(* CoDeSys 2.3.9.41 project: phase 8e.pro *)
(* Libraries: TcpIp.lib 21.3.13 08:03:14, TcBase.lib 14.5.09 12:14:08, TcSystem.lib 27.2.12 15:08:36, TcBaseMath.lib 27.7.04 12:07:56, TcMath.lib 23.9.04 15:15:30, TcMC2.lib 22.11.13 16:10:22, STANDARD.LIB 5.6.98 12:03:02, TcNC.lib 10.10.08 17:55:34, TcUtilities.lib 10.1.13 20:12:12, SysLibTargetVisu.lib 16.6.08 16:24:26, SysLibVisu.lib 7.7.04 18:17:22 *)

(* Task configuration *)
TASK Standard (PRIORITY := 1, INTERVAL := T#5ms);
	MAIN
END_TASK
TASK Fast (PRIORITY := 0, INTERVAL := T#1ms);
	MainFast();
END_TASK

(* Global variable list: Globale_Variablen *)
VAR_GLOBAL CONSTANT
	MAX_CSV_ROWS 			: UDINT := 150;
	MAX_CSV_COLUMNS 		: UDINT := 8;
	MAX_CSV_FIELD_LENGTH	: UDINT := 8;

END_VAR

VAR_GLOBAL
	FILEDATA1: ARRAY[0..MAX_CSV_ROWS, 0..MAX_CSV_COLUMNS ] OF STRING;
	trigger1: BOOL;			(* motor running*)
	trigger2: BOOL;			(* in velocity*)
	trigger3:BOOL;			(* vehicle moving*)
	encoderX:	ARRAY[1..6] OF		LREAL;
	encoderY:	ARRAY[1..6] OF		LREAL;
	heading:		ARRAY[1..6] OF		LREAL;
	headingA: LREAL;
	reset:		BOOL;
	home: BOOL;
	combinedX: LREAL;
	combinedY: LREAL;
	combinedH: LREAL;
(*for ROS*)
	robotPosX:	LREAL;
	robotPosY:	LREAL;
	robotPosTheta:	LREAL;
	robotVelX:	LREAL;
	robotVelY:	LREAL;
	robotVelTheta:	LREAL;
(*
###################
	TwinCAT NC Achsen
###################
*)


	Axis1 : AXIS_REF;
	PowerAxis1: MC_Power;
	MoveAxis1: MC_MoveVelocity;
	MoveAxis12: MC_MoveVelocity;
	ResetAxis1: MC_Reset;		(* debug function block output data *)
	HaltAxis1: MC_Halt;

	Axis2 : AXIS_REF;
	PowerAxis2: MC_Power;
	MoveAxis2: MC_MoveVelocity;
	MoveAxis22: MC_MoveVelocity;
	ResetAxis2: MC_Reset;		(* debug function block output data *)
	HaltAxis2: MC_Halt;

	Axis3 : AXIS_REF;
	PowerAxis3: MC_Power;
	MoveAxis3: MC_MoveVelocity;
	MoveAxis32: MC_MoveVelocity;
	ResetAxis3: MC_Reset;		(* debug function block output data *)
	HaltAxis3: MC_Halt;

	Axis4 : AXIS_REF;
	PowerAxis4: MC_Power;
	MoveAxis4: MC_MoveVelocity;
	MoveAxis42: MC_MoveVelocity;
	ResetAxis4: MC_Reset;		(* debug function block output data *)
	HaltAxis4: MC_Halt;


	LOCrobotPosX: LREAL;
	LOCrobotPosY: LREAL;
	LOCrobotPosTheta: LREAL;
	LOCrobotVelX: LREAL;
	LOCrobotVelY: LREAL;
	LOCrobotVelTheta: LREAL;
END_VAR

(* Global variable list: TwinCAT_Configuration *)
(* Generated automatically by TwinCAT - (read only) *)
VAR_CONFIG
	MainFast.fblocalization.encoder1.PlcToNc AT %QB1156 : PLCTONC_AXIS_REF;	(*  ~ {LinkedWith:TINC^NC-Task 1 SAF^Axes^encoder1^Inputs^encoder1_FromPlc} *)
	MainFast.fblocalization.encoder1.NcToPlc AT %IB1152 : NCTOPLC_AXIS_REF;	(*  ~ {LinkedWith:TINC^NC-Task 1 SAF^Axes^encoder1^Outputs^encoder1_ToPlc} *)
	MainFast.fblocalization.encoder2.PlcToNc AT %QB1284 : PLCTONC_AXIS_REF;	(*  ~ {LinkedWith:TINC^NC-Task 1 SAF^Axes^encoder2^Inputs^encoder2_FromPlc} *)
	MainFast.fblocalization.encoder2.NcToPlc AT %IB1280 : NCTOPLC_AXIS_REF;	(*  ~ {LinkedWith:TINC^NC-Task 1 SAF^Axes^encoder2^Outputs^encoder2_ToPlc} *)
	MainFast.fblocalization.encoder3.PlcToNc AT %QB1412 : PLCTONC_AXIS_REF;	(*  ~ {LinkedWith:TINC^NC-Task 1 SAF^Axes^encoder3^Inputs^encoder3_FromPlc} *)
	MainFast.fblocalization.encoder3.NcToPlc AT %IB1408 : NCTOPLC_AXIS_REF;	(*  ~ {LinkedWith:TINC^NC-Task 1 SAF^Axes^encoder3^Outputs^encoder3_ToPlc} *)
	MainFast.fblocalization.encoder4.PlcToNc AT %QB1540 : PLCTONC_AXIS_REF;	(*  ~ {LinkedWith:TINC^NC-Task 1 SAF^Axes^encoder4^Inputs^encoder4_FromPlc} *)
	MainFast.fblocalization.encoder4.NcToPlc AT %IB1536 : NCTOPLC_AXIS_REF;	(*  ~ {LinkedWith:TINC^NC-Task 1 SAF^Axes^encoder4^Outputs^encoder4_ToPlc} *)
	.Axis1.PlcToNc AT %QB1668 : PLCTONC_AXIS_REF;	(*  ~ {LinkedWith:TINC^NC-Task 1 SAF^Axes^motor 1^Inputs^motor 1_FromPlc} *)
	.Axis1.NcToPlc AT %IB1664 : NCTOPLC_AXIS_REF;	(*  ~ {LinkedWith:TINC^NC-Task 1 SAF^Axes^motor 1^Outputs^motor 1_ToPlc} *)
	.Axis2.PlcToNc AT %QB1796 : PLCTONC_AXIS_REF;	(*  ~ {LinkedWith:TINC^NC-Task 1 SAF^Axes^motor 2^Inputs^motor 2_FromPlc} *)
	.Axis2.NcToPlc AT %IB1792 : NCTOPLC_AXIS_REF;	(*  ~ {LinkedWith:TINC^NC-Task 1 SAF^Axes^motor 2^Outputs^motor 2_ToPlc} *)
	.Axis3.PlcToNc AT %QB1924 : PLCTONC_AXIS_REF;	(*  ~ {LinkedWith:TINC^NC-Task 1 SAF^Axes^motor 3^Inputs^motor 3_FromPlc} *)
	.Axis3.NcToPlc AT %IB1920 : NCTOPLC_AXIS_REF;	(*  ~ {LinkedWith:TINC^NC-Task 1 SAF^Axes^motor 3^Outputs^motor 3_ToPlc} *)
	.Axis4.PlcToNc AT %QB2052 : PLCTONC_AXIS_REF;	(*  ~ {LinkedWith:TINC^NC-Task 1 SAF^Axes^motor 4^Inputs^motor 4_FromPlc} *)
	.Axis4.NcToPlc AT %IB2048 : NCTOPLC_AXIS_REF;	(*  ~ {LinkedWith:TINC^NC-Task 1 SAF^Axes^motor 4^Outputs^motor 4_ToPlc} *)
END_VAR

(* Data type *)
TYPE MoveState_NC :
(
	NC_INIT,
	NC_ENABLE,
	NC_MOVE,
	NC_MOVENEXT,
	NC_ERROR,
	NC_RESET
);
END_TYPE

(* POU MAIN, ST *)
PROGRAM MAIN
VAR
	fbPLC_Reset: PLC_Reset;
	fbPLC_Start: PLC_Start;
	state_NC: MoveState_NC;
	Manual: BOOL := FALSE;
	bEnable: BOOL; (* gibt die Achse frei *)
	bReset_Axis: BOOL; (* Reset der Achse *)
	bAxis_Ready: ARRAY[1..5] OF	BOOL; (* Checks whether the axis is ready *)
	trigger2bypass: ARRAY[1..4] OF	BOOL;
	bMoveCombination: ARRAY[1..10] OF		BOOL; (* the combined movement *)
	i: INT;
	MotionReq: BOOL;
	timeToMove: TIME;
	directionToMove: INT;
	timeToMoveReal: LREAL;
	speedToMove: LREAL := 603;
	timeUp: BOOL;
	timerOn: BOOL;
	fbTON1: TON;
	myROS_connect_receiveData: ROS_connect_receiveData;
	myROS_connect_sendData: ROS_connect_sendData;
	myROS_disconnect: ROS_disconnect;
	myROS_receiveData: ROS_receiveData;
	myROS_sendData: ROS_sendData;
	myROS_convertSendData: ROS_convertSendData;
	ROS_tcpSocketReceiveData: T_HSOCKET;
	ROS_connectionOpenReceiveData: BOOL := FALSE;
	ROS_tcpSocketSendData: T_HSOCKET;
	ROS_connectionOpenSendData: BOOL := FALSE;
	ROS_closeConnection: BOOL := TRUE;
	ROS_velAxis1: LREAL := 0;
	ROS_velAxis2: LREAL := 0;
	ROS_velAxis3: LREAL := 0;
	ROS_velAxis4: LREAL := 0;
	ROS_RobotPosX: LREAL := 0;
	ROS_RobotPosY: LREAL := 0;
	ROS_RobotPosTheta: LREAL := 0;
	ROS_RobotVelX: LREAL := 0;
	ROS_RobotVelY: LREAL := 0;
	ROS_RobotVelTheta: LREAL := 0;
	sendBufferREAL: LREAL := 0;
	sendBuffer: STRING;
	sendTakt: LREAL := 0;
	vel_last1: LREAL;
	vel_current1: LREAL;
	vel_last2: LREAL;
	vel_current2: LREAL;
	vel_last3: LREAL;
	vel_current3: LREAL;
	vel_last4: LREAL;
	vel_current4: LREAL;
	startTimer1: BOOL;
	timer1On: BOOL;
	firstStart: BOOL;
	Q: BOOL;
	startPLC: BOOL;
	oldSpeedX: LREAL;
	oldSpeedY: LREAL;
	oldSpeedH: LREAL;
	connectJs: jsConnect;
	disconnectJs: jsDisconnect;
	receiveJsData: jsReceiveData;
	tcpSockeJst: T_HSOCKET;
	connectionOpen_js: BOOL := FALSE;
	closeConnection_js: BOOL := TRUE;
	XAxis: LREAL;
	YAxis: LREAL;
	ZAxis: LREAL;
	botton: LREAL;
	t1: INT;
	Name: BOOL;
END_VAR
(*
##
## This code was built by Theng Chua and Christian Scheifele, University of Stuttgart, 2014.
## It contains complete segments from Chris Jarrett, Auckland University, 2014
## and is derived in part from the TCP/IP server example on www.beckhoff.com
##
*)
(*IF (trigger3 = TRUE) THEN t1:=1; ELSE t1:=0; END_IF*)

(*
###################
Manual
###################
*)
IF (Manual=TRUE) THEN
	IF (reset=TRUE) THEN
	fbPLC_Reset(port:=801,RESET:=TRUE);
	fbPLC_Start(port:=801,start:=TRUE);
	(*set all globle variable to zero*)
	trigger1:=FALSE;
	trigger2:=FALSE;
	trigger3:=FALSE;
	home:= TRUE;
	combinedX:=0;
	combinedY:=0;
	combinedH:=0;
	END_IF

	FOR i:=1 TO 10 BY 1 DO
		IF(bMoveCombination[i]) THEN
			directionToMove:=i;
			MotionReq:=TRUE;
		END_IF
	END_FOR

	IF(MotionReq=TRUE) THEN
		CASE directionToMove OF
		1:	ROS_velAxis1:= -speedToMove;
			ROS_velAxis2:= 0;
			ROS_velAxis3:= 0;
			ROS_velAxis4:= -speedToMove;
		2:	ROS_velAxis1:= -speedToMove;
			ROS_velAxis2:= -speedToMove;
			ROS_velAxis3:= -speedToMove;
			ROS_velAxis4:= -speedToMove;
		3:	ROS_velAxis1:= 0;
			ROS_velAxis2:= -speedToMove;
			ROS_velAxis3:= -speedToMove;
			ROS_velAxis4:= 0;
		4:	ROS_velAxis1:= -speedToMove;
			ROS_velAxis2:= speedToMove;
			ROS_velAxis3:= speedToMove;
			ROS_velAxis4:= -speedToMove;
		5:	ROS_velAxis1:= speedToMove;
			ROS_velAxis2:= -speedToMove;
			ROS_velAxis3:= -speedToMove;
			ROS_velAxis4:= speedToMove;
		6:	ROS_velAxis1:= 0;
			ROS_velAxis2:= speedToMove;
			ROS_velAxis3:= speedToMove;
			ROS_velAxis4:= 0;
		7:	ROS_velAxis1:= speedToMove;
			ROS_velAxis2:= speedToMove;
			ROS_velAxis3:= speedToMove;
			ROS_velAxis4:= speedToMove;
		8:	ROS_velAxis1:= speedToMove;
			ROS_velAxis2:= 0;
			ROS_velAxis3:= 0;
			ROS_velAxis4:= speedToMove;
		9:	ROS_velAxis1:= -speedToMove;
			ROS_velAxis2:= speedToMove;
			ROS_velAxis3:= -speedToMove;
			ROS_velAxis4:= speedToMove;
		10:	ROS_velAxis1:= speedToMove;
			ROS_velAxis2:= -speedToMove;
			ROS_velAxis3:= speedToMove;
			ROS_velAxis4:= -speedToMove;
		ELSE
			ROS_velAxis1:= 0;
			ROS_velAxis2:= 0;
			ROS_velAxis3:= 0;
			ROS_velAxis4:= 0;
		END_CASE
	timetomove:= REAL_TO_TIME (timeToMoveReal);
	timerOn:=TRUE;
	END_IF

	fbTON1(IN:=timerOn, PT:=timeToMove, Q=>timeUp, ET=>);

	IF (timeUp=TRUE)  THEN
	MotionReq:=FALSE;
	bMoveCombination[directionToMove]:=FALSE;
	ROS_velAxis1:= 0;
	ROS_velAxis2:= 0;
	ROS_velAxis3:= 0;
	ROS_velAxis4:= 0;
	directionToMove:=0;
	timerOn:=FALSE;
	END_IF
(*
###################
ODOMETRY
###################
*) (* trigger 1 and trigger 2*)
	IF (vel_current1<>0 OR vel_current2<>0 OR vel_current3<>0 OR vel_current4<>0) THEN trigger1:=TRUE;
	ELSE trigger1:=FALSE;
	END_IF
	IF (trigger1) THEN  trigger2bypass[1]:=FALSE; trigger2bypass[2]:=FALSE; trigger2bypass[3]:=FALSE; trigger2bypass[4]:=FALSE;
		IF (vel_current1=0) THEN trigger2bypass[1]:=TRUE; END_IF
		IF (vel_current2=0) THEN trigger2bypass[2]:=TRUE;END_IF
		IF (vel_current3=0) THEN trigger2bypass[3]:=TRUE;END_IF
		IF (vel_current4=0) THEN trigger2bypass[4]:=TRUE;END_IF
	END_IF
	trigger2 := (MoveAxis1.InVelocity OR trigger2bypass[1]) AND (MoveAxis2.InVelocity OR trigger2bypass[2]) AND (MoveAxis3.InVelocity OR trigger2bypass[3]) AND (MoveAxis4.InVelocity OR trigger2bypass[4])
			OR  (MoveAxis12.InVelocity OR trigger2bypass[1]) AND (MoveAxis22.InVelocity OR trigger2bypass[2]) AND (MoveAxis32.InVelocity OR trigger2bypass[3]) AND (MoveAxis42.InVelocity OR trigger2bypass[4]);

ELSE  (* after this run on auto*)

(*###################
ROS TCP/IP CONNECTION
###################

Close TCP port from last time-remove after DEBUG*)

		IF ROS_closeConnection THEN
		myROS_disconnect(bCloseAll:=ROS_closeConnection);
		ROS_closeConnection:=FALSE;
		END_IF

		(*Open a connection to ROS - Receive Data*)
		IF NOT ROS_connectionOpenReceiveData THEN
		myROS_connect_receiveData(RosConnected=>ROS_connectionOpenReceiveData, socketToUse=>ROS_tcpSocketReceiveData);
		END_IF
		IF ROS_connectionOpenReceiveData THEN
		myROS_receiveData(socketToUse:=ROS_tcpSocketReceiveData,velAxis1=>ROS_velAxis1, velAxis2=>ROS_velAxis2, velAxis3=>ROS_velAxis3, velAxis4=>ROS_velAxis4);
		END_IF

		(*Open a connection to ROS - Send Data*)
		IF NOT ROS_connectionOpenSendData THEN
		myROS_connect_sendData(RosConnected=>ROS_connectionOpenSendData, socketToUse=>ROS_tcpSocketSendData);
		END_IF

		(*ODOMETRY SORCE*)
		ROS_RobotPosX := LOCrobotPosY;
		ROS_RobotPosY := LOCrobotPosX;
		ROS_RobotPosTheta :=  LOCrobotPosTheta;
		ROS_RobotVelX :=  LOCrobotVelX;
		ROS_RobotVelY :=  LOCrobotVelY;
		ROS_RobotVelTheta :=  LOCrobotVelTheta;

		IF ROS_connectionOpenSendData THEN
		(* TAKTZEIT EINSTELLEN *)
		sendTakt := sendTakt + 0.1;
			IF sendTakt > 1THEN
			myROS_convertSendData(robotPosX:=ROS_RobotPosX, robotPosY:=ROS_RobotPosY, robotPosTheta:= ROS_RobotPosTheta, robotVelX:=ROS_RobotVelX, robotVelY:=ROS_RobotVelY, robotVelTheta:=ROS_RobotVelTheta, send_message=>sendBuffer );
			myROS_sendData(sendBuffer:=sendBuffer, socketToUse:=ROS_tcpSocketSendData);
			sendTakt := 0;
			END_IF
		END_IF


END_IF (* for manual running*)

(*
###################
TwinCAT NC Achsen
###################
*)
Axis1.ReadStatus;
Axis2.ReadStatus;
Axis3.ReadStatus;
Axis4.ReadStatus;

vel_current1 := -ROS_velAxis1;
vel_current2 := ROS_velAxis2;
vel_current3 := -ROS_velAxis3;
vel_current4 := ROS_velAxis4;

(* move axis using a state machine *)
CASE state_NC OF
		NC_INIT :	(* initialisation *)
			(* initialize all function blocks *)
			MoveAxis1.Execute := FALSE;
			ResetAxis1.Execute := FALSE;
			MoveAxis2.Execute := FALSE;
			ResetAxis2.Execute := FALSE;
			MoveAxis3.Execute := FALSE;
			ResetAxis3.Execute := FALSE;
			MoveAxis4.Execute := FALSE;
			ResetAxis4.Execute := FALSE;
			MoveAxis12.Execute := FALSE;
			MoveAxis22.Execute := FALSE;
			MoveAxis32.Execute := FALSE;
			MoveAxis42.Execute := FALSE;
			HaltAxis1.Execute := FALSE;
			HaltAxis2.Execute := FALSE;
			HaltAxis3.Execute := FALSE;
			HaltAxis4.Execute := FALSE;

			state_NC := NC_ENABLE;

		NC_ENABLE :
			PowerAxis1.Enable := TRUE;
			PowerAxis1.Enable_Positive := TRUE;
			PowerAxis1.Enable_Negative := TRUE;
			PowerAxis2.Enable := TRUE;
			PowerAxis2.Enable_Positive := TRUE;
			PowerAxis2.Enable_Negative := TRUE;
			PowerAxis3.Enable := TRUE;
			PowerAxis3.Enable_Positive := TRUE;
			PowerAxis3.Enable_Negative := TRUE;
			PowerAxis4.Enable := TRUE;
			PowerAxis4.Enable_Positive := TRUE;
			PowerAxis4.Enable_Negative := TRUE;

			IF PowerAxis1.Status AND PowerAxis2.Status AND PowerAxis3.Status AND PowerAxis4.Status THEN
				state_NC := NC_MOVE;
			ELSIF PowerAxis1.Error AND PowerAxis2.Error AND PowerAxis3.Error AND PowerAxis4.Error THEN
				state_NC := NC_ERROR;
			END_IF

		NC_MOVE :
			IF vel_current1>0 THEN
				HaltAxis1.Execute := FALSE;
				MoveAxis1.Direction := MC_Positive_Direction;
				MoveAxis1.Velocity := vel_current1;
				MoveAxis1.BufferMode := MC_Aborting;
				MoveAxis1.Execute := TRUE;
			ELSIF vel_current1<0 THEN
				HaltAxis1.Execute := FALSE;
				MoveAxis1.Direction := MC_Negative_Direction;
				MoveAxis1.Velocity := -vel_current1;
				MoveAxis1.BufferMode := MC_Aborting;
				MoveAxis1.Execute := TRUE;
			ELSE
				HaltAxis1.BufferMode := MC_Aborting;
				HaltAxis1.Execute := TRUE;
			END_IF;


			IF vel_current2>0 THEN
				HaltAxis2.Execute := FALSE;
				MoveAxis2.Direction := MC_Positive_Direction;
				MoveAxis2.Velocity := vel_current2;
				MoveAxis2.BufferMode := MC_Aborting;
				MoveAxis2.Execute := TRUE;
			ELSIF vel_current2<0 THEN
				HaltAxis2.Execute := FALSE;
				MoveAxis2.Direction := MC_Negative_Direction;
				MoveAxis2.Velocity := -vel_current2;
				MoveAxis2.BufferMode := MC_Aborting;
				MoveAxis2.Execute := TRUE;
			ELSE
				HaltAxis2.BufferMode := MC_Aborting;
				HaltAxis2.Execute := TRUE;
			END_IF;


			IF vel_current3>0 THEN
				HaltAxis3.Execute := FALSE;
				MoveAxis3.Direction := MC_Positive_Direction;
				MoveAxis3.Velocity := vel_current3;
				MoveAxis3.BufferMode := MC_Aborting;
				MoveAxis3.Execute := TRUE;
			ELSIF vel_current3<0 THEN
				HaltAxis3.Execute := FALSE;
				MoveAxis3.Direction := MC_Negative_Direction;
				MoveAxis3.Velocity := -vel_current3;
				MoveAxis3.BufferMode := MC_Aborting;
				MoveAxis3.Execute := TRUE;
			ELSE
				HaltAxis3.BufferMode := MC_Aborting;
				HaltAxis3.Execute := TRUE;
			END_IF;


			IF vel_current4>0 THEN
				HaltAxis4.Execute := FALSE;
				MoveAxis4.Direction := MC_Positive_Direction;
				MoveAxis4.Velocity := vel_current4;
				MoveAxis4.BufferMode := MC_Aborting;
				MoveAxis4.Execute := TRUE;
			ELSIF vel_current4<0 THEN
				HaltAxis4.Execute := FALSE;
				MoveAxis4.Direction := MC_Negative_Direction;
				MoveAxis4.Velocity := -vel_current4;
				MoveAxis4.BufferMode := MC_Aborting;
				MoveAxis4.Execute := TRUE;
			ELSE
				HaltAxis4.BufferMode := MC_Aborting;
				HaltAxis4.Execute := TRUE;
			END_IF;

			IF vel_last1<>vel_current1 OR vel_last2<>vel_current2 OR vel_last3<>vel_current3 OR vel_last4<>vel_current4 THEN
				MoveAxis1.Execute := FALSE;
				MoveAxis2.Execute := FALSE;
				MoveAxis3.Execute := FALSE;
				MoveAxis4.Execute := FALSE;
				vel_last1 := vel_current1;
				vel_last2 := vel_current2;
				vel_last3 := vel_current3;
				vel_last4 := vel_current4;
				state_NC := NC_MOVENEXT;
			END_IF;
			IF  MoveAxis1.CommandAborted OR MoveAxis1.Error OR MoveAxis2.CommandAborted OR MoveAxis2.Error OR MoveAxis3.CommandAborted OR MoveAxis3.Error OR MoveAxis4.CommandAborted OR MoveAxis4.Error THEN
				state_NC := NC_MOVE;
			END_IF

		NC_MOVENEXT :
			IF vel_current1>0 THEN
				HaltAxis1.Execute := FALSE;
				MoveAxis12.Direction := MC_Positive_Direction;
				MoveAxis12.Velocity := vel_current1;
				MoveAxis12.BufferMode := MC_Aborting;
				MoveAxis12.Execute := TRUE;
			ELSIF vel_current1<0 THEN
				HaltAxis1.Execute := FALSE;
				MoveAxis12.Direction := MC_Negative_Direction;
				MoveAxis12.Velocity := -vel_current1;
				MoveAxis12.BufferMode := MC_Aborting;
				MoveAxis12.Execute := TRUE;
			ELSE
				HaltAxis1.BufferMode := MC_Aborting;
				HaltAxis1.Execute := TRUE;
			END_IF;


			IF vel_current2>0 THEN
				HaltAxis2.Execute := FALSE;
				MoveAxis22.Direction := MC_Positive_Direction;
				MoveAxis22.Velocity := vel_current2;
				MoveAxis22.BufferMode := MC_Aborting;
				MoveAxis22.Execute := TRUE;
			ELSIF vel_current2<0 THEN
				HaltAxis2.Execute := FALSE;
				MoveAxis22.Direction := MC_Negative_Direction;
				MoveAxis22.Velocity := -vel_current2;
				MoveAxis22.BufferMode := MC_Aborting;
				MoveAxis22.Execute := TRUE;
			ELSE
				HaltAxis2.BufferMode := MC_Aborting;
				HaltAxis2.Execute := TRUE;
			END_IF;


			IF vel_current3>0 THEN
				HaltAxis3.Execute := FALSE;
				MoveAxis32.Direction := MC_Positive_Direction;
				MoveAxis32.Velocity := vel_current3;
				MoveAxis32.BufferMode := MC_Aborting;
				MoveAxis32.Execute := TRUE;
			ELSIF vel_current3<0 THEN
				HaltAxis3.Execute := FALSE;
				MoveAxis32.Direction := MC_Negative_Direction;
				MoveAxis32.Velocity := -vel_current3;
				MoveAxis32.BufferMode := MC_Aborting;
				MoveAxis32.Execute := TRUE;
			ELSE
				HaltAxis3.BufferMode := MC_Aborting;
				HaltAxis3.Execute := TRUE;
			END_IF;


			IF vel_current4>0 THEN
				HaltAxis4.Execute := FALSE;
				MoveAxis42.Direction := MC_Positive_Direction;
				MoveAxis42.Velocity := vel_current4;
				MoveAxis42.BufferMode := MC_Aborting;
				MoveAxis42.Execute := TRUE;
			ELSIF vel_current4<0 THEN
				HaltAxis4.Execute := FALSE;
				MoveAxis42.Direction := MC_Negative_Direction;
				MoveAxis42.Velocity := -vel_current4;
				MoveAxis42.BufferMode := MC_Aborting;
				MoveAxis42.Execute := TRUE;
			ELSE
				HaltAxis4.BufferMode := MC_Aborting;
				HaltAxis4.Execute := TRUE;
			END_IF;

			IF vel_last1<>vel_current1 OR vel_last2<>vel_current2 OR vel_last3<>vel_current3 OR vel_last4<>vel_current4 THEN
				MoveAxis12.Execute := FALSE;
				MoveAxis22.Execute := FALSE;
				MoveAxis32.Execute := FALSE;
				MoveAxis42.Execute := FALSE;
				vel_last1 := vel_current1;
				vel_last2 := vel_current2;
				vel_last3 := vel_current3;
				vel_last4 := vel_current4;
				state_NC := NC_MOVE;
			END_IF;
			IF  MoveAxis12.CommandAborted OR MoveAxis12.Error OR MoveAxis22.CommandAborted OR MoveAxis22.Error OR MoveAxis32.CommandAborted OR MoveAxis32.Error OR MoveAxis42.CommandAborted OR MoveAxis42.Error THEN
				state_NC := NC_MOVE;
			END_IF


		NC_ERROR :
			IF Axis1.Status.Error OR Axis2.Status.Error OR Axis3.Status.Error OR Axis4.Status.Error THEN
				state_NC := NC_RESET;	(* axis error requires reset *)
			ELSE
				state_NC := NC_INIT;		(* function block errors don't need a reset *)
			END_IF

		NC_RESET :
			ResetAxis1.Execute := TRUE;
			ResetAxis2.Execute := TRUE;
			ResetAxis3.Execute := TRUE;
			ResetAxis4.Execute := TRUE;
			IF ResetAxis1.Done AND ResetAxis2.Done AND ResetAxis3.Done AND ResetAxis4.Done THEN
				state_NC := NC_INIT;
			ELSIF ResetAxis1.Error OR ResetAxis2.Error OR ResetAxis3.Error OR ResetAxis4.Error THEN
				state_NC := NC_INIT; (* can't do anything here *)
			END_IF

END_CASE

ActPower;	(* call the power function block *)
ActMove;	(* call the move function block *)
ActReset;	(* call the reset function block *)
ActHaltAxis1;
ActHaltAxis2;
ActHaltAxis3;
ActHaltAxis4;
END_PROGRAM
ACTION ActHaltAxis1:
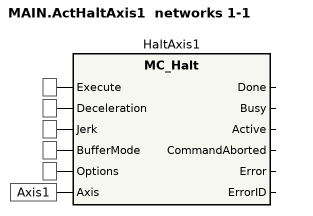
_FBD_ (* Function Block Diagram *)
NETWORK 1
	HaltAxis1:MC_Halt(Execute: , Deceleration: , Jerk: , BufferMode: , Options: , Axis: Axis1)
_END_FBD_
END_ACTION
ACTION ActHaltAxis2:
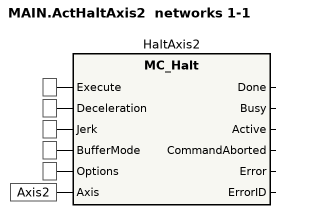
_FBD_ (* Function Block Diagram *)
NETWORK 1
	HaltAxis2:MC_Halt(Execute: , Deceleration: , Jerk: , BufferMode: , Options: , Axis: Axis2)
_END_FBD_
END_ACTION
ACTION ActHaltAxis3:
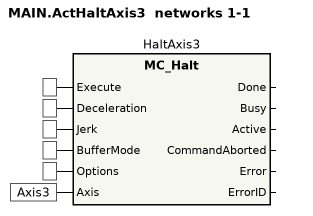
_FBD_ (* Function Block Diagram *)
NETWORK 1
	HaltAxis3:MC_Halt(Execute: , Deceleration: , Jerk: , BufferMode: , Options: , Axis: Axis3)
_END_FBD_
END_ACTION
ACTION ActHaltAxis4:
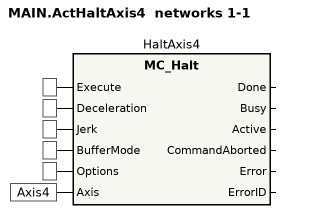
_FBD_ (* Function Block Diagram *)
NETWORK 1
	HaltAxis4:MC_Halt(Execute: , Deceleration: , Jerk: , BufferMode: , Options: , Axis: Axis4)
_END_FBD_
END_ACTION
ACTION ActMove:
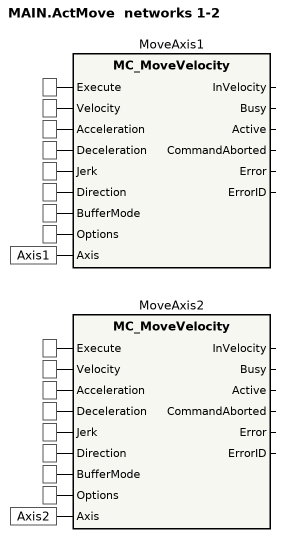
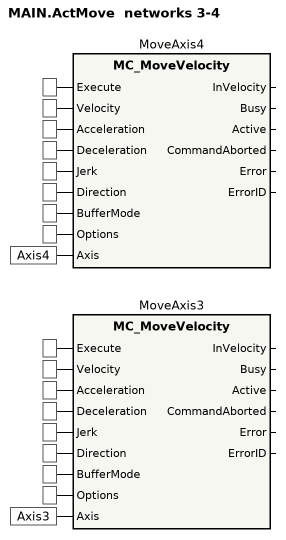
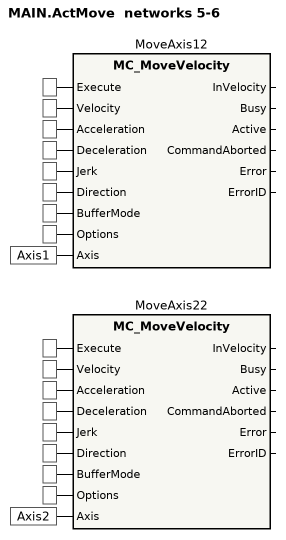
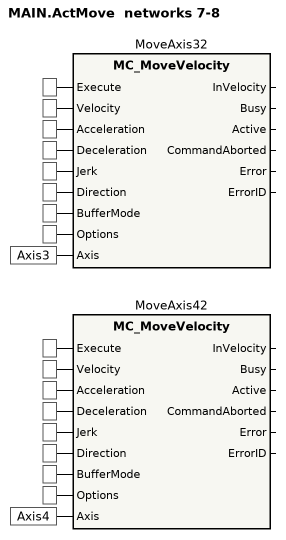
_FBD_ (* Function Block Diagram *)
NETWORK 1
	MoveAxis1:MC_MoveVelocity(Execute: , Velocity: , Acceleration: , Deceleration: , Jerk: , Direction: , BufferMode: , Options: , Axis: Axis1)
NETWORK 2
	MoveAxis2:MC_MoveVelocity(Execute: , Velocity: , Acceleration: , Deceleration: , Jerk: , Direction: , BufferMode: , Options: , Axis: Axis2)
NETWORK 3
	MoveAxis4:MC_MoveVelocity(Execute: , Velocity: , Acceleration: , Deceleration: , Jerk: , Direction: , BufferMode: , Options: , Axis: Axis4)
NETWORK 4
	MoveAxis3:MC_MoveVelocity(Execute: , Velocity: , Acceleration: , Deceleration: , Jerk: , Direction: , BufferMode: , Options: , Axis: Axis3)
NETWORK 5
	MoveAxis12:MC_MoveVelocity(Execute: , Velocity: , Acceleration: , Deceleration: , Jerk: , Direction: , BufferMode: , Options: , Axis: Axis1)
NETWORK 6
	MoveAxis22:MC_MoveVelocity(Execute: , Velocity: , Acceleration: , Deceleration: , Jerk: , Direction: , BufferMode: , Options: , Axis: Axis2)
NETWORK 7
	MoveAxis32:MC_MoveVelocity(Execute: , Velocity: , Acceleration: , Deceleration: , Jerk: , Direction: , BufferMode: , Options: , Axis: Axis3)
NETWORK 8
	MoveAxis42:MC_MoveVelocity(Execute: , Velocity: , Acceleration: , Deceleration: , Jerk: , Direction: , BufferMode: , Options: , Axis: Axis4)
_END_FBD_
END_ACTION
ACTION ActPower:
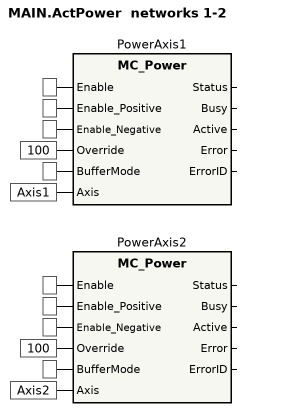
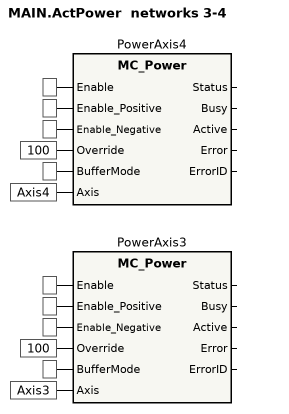
_FBD_ (* Function Block Diagram *)
NETWORK 1
	PowerAxis1:MC_Power(Enable: , Enable_Positive: , Enable_Negative: , Override: 100, BufferMode: , Axis: Axis1)
NETWORK 2
	PowerAxis2:MC_Power(Enable: , Enable_Positive: , Enable_Negative: , Override: 100, BufferMode: , Axis: Axis2)
NETWORK 3
	PowerAxis4:MC_Power(Enable: , Enable_Positive: , Enable_Negative: , Override: 100, BufferMode: , Axis: Axis4)
NETWORK 4
	PowerAxis3:MC_Power(Enable: , Enable_Positive: , Enable_Negative: , Override: 100, BufferMode: , Axis: Axis3)
_END_FBD_
END_ACTION
ACTION ActReset:
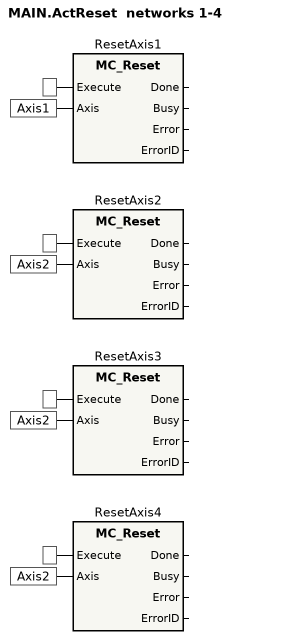
_FBD_ (* Function Block Diagram *)
NETWORK 1
	ResetAxis1:MC_Reset(Execute: , Axis: Axis1)
NETWORK 2
	ResetAxis2:MC_Reset(Execute: , Axis: Axis2)
NETWORK 3
	ResetAxis3:MC_Reset(Execute: , Axis: Axis2)
NETWORK 4
	ResetAxis4:MC_Reset(Execute: , Axis: Axis2)
_END_FBD_
END_ACTION

(* POU ROS_connect_receiveData, ST *)
FUNCTION_BLOCK ROS_connect_receiveData
VAR


	(*Functions*)
	openSocket: BOOL:=FALSE;
	fb_listen: FB_SocketListen;
	fb_accept: FB_SocketAccept;
	(*Timers*)
	fbAcceptTON: TON;

	(*TCP socket variables*)
	activeSocketHandle: T_HSOCKET;
	socketHandle: T_HSOCKET;



	(*Error variables*)
	listenError: UDINT:=0;
	acceptError: UDINT;
	listenErrSet: BOOL;
	closeError: UDINT;
	sendError: UDINT;
	receiveError: UDINT;
	bSendError: BOOL;


	(*Trigger Variables*)
	bCloseAll: BOOL := TRUE;

	(*Connection information*)
	portNumber: INT:=711;
	bAccepted: BOOL;

	(*Constants*)
	PLCPRJ_ACCEPT_POLLING_TIME: TIME:=T#1s;

	display: LREAL;
	heading: LREAL;

	state: INT:=0;

	xDist: LREAL;
	yDist: LREAL;
	zDist: LREAL;


	listening: BOOL;
END_VAR
VAR_OUTPUT
	RosConnected: BOOL;
	socketToUse: T_HSOCKET;
END_VAR
(*
##
## This code was built by Christian Scheifele, University of Stuttgart, 2014.
## It contains complete segments from Chris Jarrett, Auckland University, 2014
## and is derived in part from the TCP/IP server example on www.beckhoff.com
##
*)

CASE state OF
0:

IF(fb_Listen.hListener.localAddr.nPort=portNumber) THEN
RETURN;

ELSE
state:=1;
END_IF

1:
fb_listen
(
	sSrvNetId:='' ,
	sLocalHost:='',
	nLocalPort:=portNumber,
	bExecute:=TRUE,
	tTimeout:=T#5s,
	hListener=>socketHandle,
	nErrId=>listenError,
	bError=>listenErrSet,

);

	IF(fb_Listen.hListener.localAddr.nPort=portNumber) THEN
		fb_listen(bExecute:=FALSE); 		(*Start listening and move to the accept state*)

		state:=2;
	ELSE
		(*Return to the listening state*)
		state:=1;
	END_IF



2:

(*Start accepting a client connection*)
fbAcceptTON( IN := TRUE, PT := T#2s);  (*Start a timer to poll for the accepted connection*)
		IF fbAcceptTON.Q THEN
			fbAcceptTON( IN := FALSE );	(*Reset timer*)
			fb_accept(  bExecute := FALSE  ); (*Generate a rising edge to activate the accept function*)
			fb_accept(hListener := socketHandle, bExecute:= TRUE, hSocket=>activeSocketHandle );
			state:=3; (*Move to the state where the client is accepted*)

			fbAcceptTON( IN := FALSE);

		END_IF
3:
(*Complete accpeting the client connection*)
	fb_accept( bExecute := FALSE ); (*Reset the accept function to try connection again if necessary*)
	IF NOT fb_accept.bBusy THEN
		IF NOT fb_accept.bError THEN
			IF fb_accept.bAccepted THEN
				bAccepted := TRUE; (*If the client connection is accepted without error then move to the send state*)
				fb_accept(bExecute:=FALSE);
				socketToUse:=fb_accept.hSocket;
				state:=4;
			ELSE
				fb_listen(bExecute:=FALSE);
				fb_accept(bExecute:=FALSE);
				RosConnected:=FALSE; (*If the connection attempt was not successful, return the boolean as false*)
				fbAcceptTON( IN := FALSE);
				state:=2;
			END_IF
		END_IF
	END_IF
4:
RosConnected:=TRUE;
RETURN;

END_CASE;
END_FUNCTION_BLOCK

(* POU ROS_connect_sendData, ST *)
FUNCTION_BLOCK ROS_connect_sendData
VAR


	(*Functions*)
	openSocket: BOOL:=FALSE;
	fb_listen: FB_SocketListen;
	fb_accept: FB_SocketAccept;
	(*Timers*)
	fbAcceptTON: TON;

	(*TCP socket variables*)
	activeSocketHandle: T_HSOCKET;
	socketHandle: T_HSOCKET;



	(*Error variables*)
	listenError: UDINT:=0;
	acceptError: UDINT;
	listenErrSet: BOOL;
	closeError: UDINT;
	sendError: UDINT;
	receiveError: UDINT;
	bSendError: BOOL;


	(*Trigger Variables*)
	bCloseAll: BOOL := TRUE;

	(*Connection information*)
	portNumber: INT:=712;
	bAccepted: BOOL;

	(*Constants*)
	PLCPRJ_ACCEPT_POLLING_TIME: TIME:=T#1s;

	display: LREAL;
	heading: LREAL;

	state: INT:=0;

	xDist: LREAL;
	yDist: LREAL;
	zDist: LREAL;


	listening: BOOL;
END_VAR
VAR_OUTPUT
	RosConnected: BOOL;
	socketToUse: T_HSOCKET;
END_VAR
(*
##
## This code was built by Christian Scheifele, University of Stuttgart, 2014.
## It contains complete segments from Chris Jarrett, Auckland University, 2014
## and is derived in part from the TCP/IP server example on www.beckhoff.com
##
*)

CASE state OF
0:

IF(fb_Listen.hListener.localAddr.nPort=portNumber) THEN
RETURN;

ELSE
state:=1;
END_IF

1:
(*This code was built by Chris Jarrett, Auckland University, 2014. It is derived in part from the TCP/IP server example on www.beckhoff.com*)
fb_listen
(
	sSrvNetId:='' ,
	sLocalHost:='',
	nLocalPort:=portNumber,
	bExecute:=TRUE,
	tTimeout:=T#5s,
	hListener=>socketHandle,
	nErrId=>listenError,
	bError=>listenErrSet,

);

	IF(fb_Listen.hListener.localAddr.nPort=portNumber) THEN
		fb_listen(bExecute:=FALSE); 		(*Start listening and move to the accept state*)

		state:=2;
	ELSE
		(*Return to the listening state*)
		state:=1;
	END_IF



2:

(*Start accepting a client connection*)
fbAcceptTON( IN := TRUE, PT := T#2s);  (*Start a timer to poll for the accepted connection*)
		IF fbAcceptTON.Q THEN
			fbAcceptTON( IN := FALSE );	(*Reset timer*)
			fb_accept(  bExecute := FALSE  ); (*Generate a rising edge to activate the accept function*)
			fb_accept(hListener := socketHandle, bExecute:= TRUE, hSocket=>activeSocketHandle );
			state:=3; (*Move to the state where the client is accepted*)

			fbAcceptTON( IN := FALSE);

		END_IF
3:
(*Complete accpeting the client connection*)
	fb_accept( bExecute := FALSE ); (*Reset the accept function to try connection again if necessary*)
	IF NOT fb_accept.bBusy THEN
		IF NOT fb_accept.bError THEN
			IF fb_accept.bAccepted THEN
				bAccepted := TRUE; (*If the client connection is accepted without error then move to the send state*)
				fb_accept(bExecute:=FALSE);
				socketToUse:=fb_accept.hSocket;
				state:=4;
			ELSE
				fb_listen(bExecute:=FALSE);
				fb_accept(bExecute:=FALSE);
				RosConnected:=FALSE; (*If the connection attempt was not successful, return the boolean as false*)
				fbAcceptTON( IN := FALSE);
				state:=2;
			END_IF
		END_IF
	END_IF
4:
RosConnected:=TRUE;
RETURN;

END_CASE;
END_FUNCTION_BLOCK

(* POU ROS_disconnect, ST *)
FUNCTION_BLOCK ROS_disconnect
VAR_INPUT
	bCloseAll: BOOL;
END_VAR
VAR_OUTPUT
	connectionClosed: BOOL;
END_VAR
VAR
	fb_closeAll: FB_SocketCloseAll;
END_VAR
(*
##
## This code was built by Christian Scheifele, University of Stuttgart, 2014.
## It contains complete segments from Chris Jarrett, Auckland University, 2014
## and is derived in part from the TCP/IP server example on www.beckhoff.com
##
*)


(*This function closes the TCP/IP port being used the ROS connection*)

IF bCloseAll THEN
	bCloseAll:=FALSE;
	(*Close all open ports*)
	fb_closeAll(sSrvNetId:='', bExecute:=TRUE, tTimeOut:=T#5s );
ELSE
	fb_closeAll(bExecute:=FALSE);
END_IF


(*Move to the listening state*)
IF NOT fb_closeAll.bError THEN
	connectionClosed:=TRUE;


ELSE
connectionClosed:=FALSE;
END_IF
RETURN;
END_FUNCTION_BLOCK

(* POU ROS_receiveData, ST *)
FUNCTION_BLOCK ROS_receiveData
VAR_INPUT
	socketToUse: T_HSOCKET;
END_VAR
VAR_OUTPUT
	dataReceived: BOOL;
	velAxis1: LREAL;
	velAxis2: LREAL;
	velAxis3: LREAL;
	velAxis4: LREAL;
END_VAR
VAR
	(*Connection timers*)
	fbReceiveTON: TON;
	fbResetTON:TON;
	reset: BOOL;
	timeup:BOOL;

 	(*Functions*)
	fb_receive: FB_SocketReceive;

	(*Send and receive data and variables*)
	receiveBuffer: ARRAY[0..27] OF BYTE;
	bytesReceived: UDINT;
	sendBuffer: STRING;
	sendBufferAddress: DWORD;
	cbReceived, startPos, endPos, idx : UDINT;
	cbFrame: UDINT;
	sFromClient: T_MaxString;
	overflow: BOOL;
	endFound: BOOL;

	(*Error variables*)
	acceptError: UDINT;
	receiveError: UDINT;

	state: INT:=1;
END_VAR
(*
##
## This code was built by Christian Scheifele, University of Stuttgart, 2014.
## It contains complete segments from Chris Jarrett, Auckland University, 2014
## and is derived in part from the TCP/IP server example on www.beckhoff.com
##
*)

CASE state OF
1:
(*Receive information*)
	fbReceiveTON(  IN := FALSE, PT:=T#0s); (*Receive first request immediately*)
	fbReceiveTON(  IN := TRUE ); (*Start a timer to ensure complete transfer of information*)

		IF fbReceiveTON.Q THEN
			fbReceiveTON(  IN := FALSE);
			fb_receive(bExecute:=FALSE);  (*Generate a rising edge to start receiving data*)
			fb_receive
			(
				sSrvNetId:='',
				hSocket :=socketToUse,
				cbLen:=SIZEOF(receiveBuffer)-cbReceived,
				pDest:=ADR(receiveBuffer)+cbReceived,
				tTimeout:=T#5s,
				nRecBytes=>bytesReceived,
				nErrId=>receiveError,
				bExecute:=TRUE,
			);

	(*Move to the receive completion state*)
	state:=2;
	END_IF

2:
(*Continue receiving data*)
	fb_receive( bExecute := FALSE );
	IF NOT fb_receive.bBusy THEN
		IF NOT fb_receive.bError THEN (*If no error has occurred then start the actual receiving of data*)

			IF (fb_receive.nRecBytes>0) THEN (*Bytes have been received*)

				startPos:=cbReceived; (*index of first data byte*)
				endPos:=cbReceived+fb_receive.nRecBytes-1; (*index of last byte*)
				cbReceived:=cbReceived+fb_receive.nRecBytes; (*Calculating the number of received data bytes*)
				cbFrame:=0; (*Reset the frame length*)


				IF cbReceived<SIZEOF(sFromClient) THEN (*no overflow*)
					fbReceiveTON(IN:=FALSE, PT:=T#0S);

					(*Search for the string delimiter(separation character for different strings)*)
					FOR idx:=startPos TO endPos BY 1 DO
						IF receiveBuffer[idx]=0 THEN (*String delimiter found*)
							cbFrame:=idx+1;(*calculate length of received string*)
							MEMCPY(ADR(sFromClient), ADR(receiveBuffer),cbFrame); (*copy the received string to the output variable*)
							MEMMOVE(ADR(receiveBuffer), ADR(receiveBuffer[cbFrame]), cbReceived-cbFrame);(*move remaining data bytes*)
							dataReceived:=TRUE;  	(*Send an acknowledgement of data received*)
							state:=3; (*Move to the receive completion state*)
							endFound:=TRUE;
							EXIT;
						END_IF
					END_FOR
				ELSE(*no more free buffer space-overflow*)

					dataReceived:=FALSE;; (*Go to error state*)
					overflow:=TRUE;
					state:=4;
				END_IF
			ELSE(*no data received*)
					fbReceiveTON(IN:=FALSE, PT:=T#0ms);
					state:=1;
			END_IF
		ELSE(*error receiving data, exit function*)
			state:=4;
			dataReceived:=FALSE;
		END_IF
	END_IF

3:
(*State used to process data*)
	velAxis1:=(STRING_TO_LREAL(MID(sFromClient, 7, 1)))/100;  (*Extract the x distance*)
	velAxis2:=(STRING_TO_LREAL(MID(sFromClient, 7, 8)))/100;
	velAxis3:=(STRING_TO_LREAL(MID(sFromClient, 7, 15)))/100;
	velAxis4:=(STRING_TO_LREAL(MID(sFromClient, 7, 22)))/100;

       (*Fixing an issue of negative numbers
	IF velAxis1 >  -100 THEN
		velAxis1:=velAxis1/10;
	END_IF
	IF velAxis2 > -100 THEN
		velAxis2:=velAxis2/10;
	END_IF
	IF velAxis3 > -100 THEN
		velAxis3:=velAxis3/10;
	END_IF
	IF velAxis4 > -100  THEN
		velAxis4:=velAxis4/10;
	END_IF*)

	fb_receive(bExecute:=FALSE); (*Reset the receive function*)
	startPos:=0; (*reset buffer beginning pointer*)
	endPos:=0;  (*reset buffer end pointer*)
	cbReceived:=0; (*reset bytes received counter*)
	sFromClient:=''; (*reset transition variable*)

	state:=1;
	RETURN;

4: (*Unused except for as an error state*)
	trigger1:=FALSE;trigger2:=TRUE;
	trigger2:=FALSE;

	velAxis1:=0;
	velAxis2:=0;
	velAxis3:=0;
	velAxis4:=0;

	(*Clear buffer-PROBABLY UNNECESSARY*)
	receiveBuffer[0]:=0;
	receiveBuffer[1]:=0;
	receiveBuffer[2]:=0;
	receiveBuffer[3]:=0;
	receiveBuffer[4]:=0;
	receiveBuffer[5]:=0;
	receiveBuffer[6]:=0;
	receiveBuffer[7]:=0;
	receiveBuffer[8]:=0;
	receiveBuffer[9]:=0;
	receiveBuffer[10]:=0;
	receiveBuffer[11]:=0;
	receiveBuffer[12]:=0;
	receiveBuffer[13]:=0;
	receiveBuffer[14]:=0;
	receiveBuffer[15]:=0;
	receiveBuffer[16]:=0;
	receiveBuffer[17]:=0;
	receiveBuffer[18]:=0;
	receiveBuffer[19]:=0;
	receiveBuffer[20]:=0;
	receiveBuffer[21]:=0;
	receiveBuffer[22]:=0;
	receiveBuffer[23]:=0;
	receiveBuffer[24]:=0;
	receiveBuffer[25]:=0;
	receiveBuffer[26]:=0;
	receiveBuffer[27]:=0;

	state:=1;
END_CASE;
END_FUNCTION_BLOCK

(* POU ROS_sendData, ST *)
FUNCTION_BLOCK ROS_sendData
VAR_INPUT
	sendBuffer: STRING;
	socketToUse: T_HSOCKET;
END_VAR
VAR_OUTPUT
END_VAR
VAR
 	(*Functions*)
	fb_send1: FB_SocketSend;
	(*Send data and variables*)
	sendBufferAddress1: DWORD;
	sendError1: UDINT;
END_VAR
(*
##
## This code was built by Christian Scheifele, University of Stuttgart, 2014.
## It  is derived in part from the TCP/IP server example on www.beckhoff.com
##
*)
	(*Send a greeting to the client*)
	sendBufferAddress1:=ADR(sendBuffer);
	(*Send information*)
	fb_send1
	(
		sSrvNetId:='',
		hSocket:=socketToUse,
		cbLen:=INT_TO_UDINT(LEN( sendBuffer ))+1,
		pSrc:=sendBufferAddress1,
		bExecute:=TRUE,
		tTimeout:=T#5s,
		nErrId=>sendError1,
	);

	fb_send1( bExecute := FALSE );
	fb_send1( bExecute := TRUE );
	fb_send1( bExecute := FALSE );
END_FUNCTION_BLOCK

(* POU ROS_convertSendData, ST *)
FUNCTION_BLOCK ROS_convertSendData
VAR_INPUT
	robotPosX: LREAL;
	robotPosY: LREAL;
	robotPosTheta: LREAL;
	robotVelX: LREAL;
	robotVelY: LREAL;
	robotVelTheta: LREAL;
END_VAR
VAR_OUTPUT
	send_message: STRING;
END_VAR
VAR
	posXString: STRING;
	posYString: STRING;
	posThetaString: STRING;
	velXString: STRING;
	velYString: STRING;
	velThetaString: STRING;
END_VAR
(*
##
## This code was built by Christian Scheifele, University of Stuttgart, 2014.
##
*)

(* Eingangsdaten verarbeiten *)
posXString := LREAL_TO_STRING(ABS(robotPosX));
posYString := LREAL_TO_STRING(ABS(robotPosY));
posThetaString := LREAL_TO_STRING(ABS(robotPosTheta)*100);
velXString := LREAL_TO_STRING(ABS(robotVelX));
velYString := LREAL_TO_STRING(ABS(robotVelY));
velThetaString := LREAL_TO_STRING(ABS(robotVelTheta)*100);

(* posXString bearbeiten *)
posXString := LEFT(posXString, FIND(posXString, '.')-1);
IF LEN(posXString) < 6 THEN
posXString := INSERT(posXString, '0000000',0 );
posXString := RIGHT(posXString, 5);
IF(robotPosX < 0) THEN
posXString := INSERT(posXString, '-',0 );
ELSE
posXString := INSERT(posXString, '0',0 );
END_IF;
END_IF;


(* posYString bearbeiten *)
posYString := LEFT(posYString, FIND(posYString, '.')-1);
IF LEN(posYString) < 7 THEN
	posYString := INSERT(posYString, '0000000',0 );
	posYString := RIGHT(posYString, 6);
	IF(robotPosY < 0) THEN
		posYString := INSERT(posYString, '-',0 );
	ELSE
		posYString := INSERT(posYString, '0',0 );
	END_IF;
END_IF;

(* posThetaString bearbeiten *)
posThetaString := LEFT(posThetaString, FIND(posThetaString, '.')-1);
IF LEN(posThetaString) < 7 THEN
	posThetaString := INSERT(posThetaString, '0000000',0 );
	posThetaString := RIGHT(posThetaString, 6);
	IF(robotPosTheta < 0) THEN
		posThetaString := INSERT(posThetaString, '-',0 );
	ELSE
		posThetaString := INSERT(posThetaString, '0',0 );
	END_IF;
END_IF;

(* velXString bearbeiten *)
velXString := LEFT(velXString, FIND(velXString, '.')-1);
IF LEN(velXString) < 7 THEN
velXString := INSERT(velXString, '0000000',0 );
velXString := RIGHT(velXString, 6);
	IF(robotVelX < 0) THEN
		velXString := INSERT(velXString, '-',0 );
	ELSE
		velXString := INSERT(velXString, '0',0 );
	END_IF;
END_IF;

(* velYString bearbeiten *)
velYString := LEFT(velYString, FIND(velYString, '.')-1);
IF LEN(velYString) < 7 THEN
velYString := INSERT(velYString, '0000000',0 );
velYString := RIGHT(velYString, 6);
	IF(robotVelY < 0) THEN
		velYString := INSERT(velYString, '-',0 );
	ELSE
		velYString := INSERT(velYString, '0',0 );
	END_IF;
END_IF;

(* velThetaString bearbeiten *)
velThetaString := LEFT(velThetaString, FIND(velThetaString, '.')-1);
IF LEN(velThetaString) < 7 THEN
velThetaString := INSERT(velThetaString, '0000000',0 );
velThetaString := RIGHT(velThetaString, 6);
	IF(robotVelTheta < 0) THEN
		velThetaString := INSERT(velThetaString, '-',0 );
	ELSE
		velThetaString := INSERT(velThetaString, '0',0 );
	END_IF;
END_IF;

send_message := CONCAT (posXString, ' ');
send_message := CONCAT (send_message, posYString);
send_message := CONCAT (send_message, ' ');
send_message := CONCAT (send_message, posThetaString);
send_message := CONCAT (send_message, ' ');
send_message := CONCAT (send_message, velXString);
send_message := CONCAT (send_message, ' ');
send_message := CONCAT (send_message, velYString);
send_message := CONCAT (send_message, ' ');
send_message := CONCAT (send_message, velThetaString);

(*send_message := '-000001 0000002 0009000 0000009 -000001 0000004';*)
END_FUNCTION_BLOCK

(* POU jsConnect, ST *)
FUNCTION_BLOCK jsConnect
VAR


	(*Functions*)
	openSocket: BOOL:=FALSE;
	fb_listen: FB_SocketListen;
	fb_accept: FB_SocketAccept;
	(*Timers*)
	fbAcceptTON: TON;

	(*TCP socket variables*)
	activeSocketHandle: T_HSOCKET;
	socketHandle: T_HSOCKET;



	(*Error variables*)
	listenError: UDINT:=0;
	acceptError: UDINT;
	listenErrSet: BOOL;
	closeError: UDINT;
	sendError: UDINT;
	receiveError: UDINT;
	bSendError: BOOL;


	(*Trigger Variables*)
	bCloseAll: BOOL := TRUE;

	(*Connection information*)
	portNumber: INT:=8880;
	bAccepted: BOOL;

	(*Constants*)
	PLCPRJ_ACCEPT_POLLING_TIME: TIME:=T#1s;

	display: LREAL;
	heading: LREAL;

	state: INT:=0;

	xDist: LREAL;
	yDist: LREAL;
	zDist: LREAL;


	listening: BOOL;
	count: INT;
	fbresetTON: TON;
	timerOn: BOOL;
	timeUp: BOOL;
END_VAR
VAR_OUTPUT
	arduinoConnected: BOOL;
	socketToUse: T_HSOCKET;
END_VAR
trigger1:=FALSE; trigger2:=FALSE;
CASE state OF
0:

IF(fb_Listen.hListener.localAddr.nPort=portNumber) THEN
RETURN;

ELSE
state:=1;
END_IF

1:
(*This code was built by Chris Jarrett, Auckland University, 2014. It is derived in part from the TCP/IP server example on www.beckhoff.com*)
(*Listening State*)
(*Open a connection*)
(*Create socket and check for errors*)

fb_listen
(
	sSrvNetId:='' ,
	sLocalHost:='',
	nLocalPort:=portNumber,
	bExecute:=TRUE,
	tTimeout:=T#5s,
	hListener=>socketHandle,
	nErrId=>listenError,
	bError=>listenErrSet,

);

	IF(fb_Listen.hListener.localAddr.nPort=portNumber) THEN
		fb_listen(bExecute:=FALSE); 		(*Start listening and move to the accept state*)

		state:=2;
	ELSE
		(*Return to the listening state*)
		state:=1;
	END_IF



2:

(*Start accepting a client connection*)
fbAcceptTON( IN := TRUE, PT := T#2s);  (*Start a timer to poll for the accepted connection*)
		IF fbAcceptTON.Q THEN
			fbAcceptTON( IN := FALSE );	(*Reset timer*)
			fb_accept(  bExecute := FALSE  ); (*Generate a rising edge to activate the accept function*)
			fb_accept(hListener := socketHandle, bExecute:= TRUE, hSocket=>activeSocketHandle );
			state:=3; (*Move to the state where the client is accepted*)

			fbAcceptTON( IN := FALSE);

		END_IF
3:
(*Complete accpeting the client connection*)
	fb_accept( bExecute := FALSE ); (*Reset the accept function to try connection again if necessary*)
	IF NOT fb_accept.bBusy THEN
		IF NOT fb_accept.bError THEN
			IF fb_accept.bAccepted THEN
				bAccepted := TRUE; (*If the client connection is accepted without error then move to the send state*)
				fb_accept(bExecute:=FALSE);
				socketToUse:=fb_accept.hSocket;

				state:=4;
			ELSE
				fb_listen(bExecute:=FALSE);
				fb_accept(bExecute:=FALSE);
				arduinoConnected:=FALSE; (*If the connection attempt was not successful, return the boolean as false*)
				fbAcceptTON( IN := FALSE);
				state:=2;

				END_IF
		END_IF
	END_IF
4:
arduinoConnected:=TRUE;
RETURN;

END_CASE;
END_FUNCTION_BLOCK

(* POU jsDisconnect, ST *)
FUNCTION_BLOCK jsDisconnect
VAR_INPUT
	bCloseAll: BOOL;
END_VAR
VAR_OUTPUT
	connectionClosed: BOOL;
END_VAR
VAR
	fb_closeAll: FB_SocketCloseAll;
END_VAR
(*This function closes the TCP/IP port being used the Arduino connection*)

IF bCloseAll THEN
	bCloseAll:=FALSE;
	(*Close all open ports*)
	fb_closeAll(sSrvNetId:='', bExecute:=TRUE, tTimeOut:=T#5s );
ELSE
	fb_closeAll(bExecute:=FALSE);
END_IF


(*Move to the listening state*)
IF NOT fb_closeAll.bError THEN
	connectionClosed:=TRUE;


ELSE
connectionClosed:=FALSE;
END_IF
RETURN;
END_FUNCTION_BLOCK

(* POU jsReceiveData, ST *)
FUNCTION_BLOCK jsReceiveData
VAR_INPUT

	socketToUse: T_HSOCKET;
END_VAR
VAR_OUTPUT
	dataReceived: BOOL;
	botton: LREAL;
	xAxis: LREAL;
	yAxis: LREAL;
	zAxis: LREAL;
END_VAR
VAR
	(*Connection timers*)
	fbReceiveTON: TON;

 	(*Functions*)
	fb_receive: FB_SocketReceive;

	(*Send and receive data and variables*)
	receiveBuffer: ARRAY[0..19] OF BYTE;
	bytesReceived: UDINT;
	sendBuffer: STRING;
	sendBufferAddress: DWORD;
	cbReceived, startPos, endPos, idx : UDINT;
	cbFrame: UDINT;
	sFromClient: T_MaxString;
	overflow: BOOL;
	endFound: BOOL;

	(*Error variables*)
	acceptError: UDINT;
	receiveError: UDINT;

	state: INT:=1;
	xAsisString: STRING;
	yAsixString: STRING;
	zAxisString: STRING;
	bottonString: STRING;
	timerOn: BOOL;
	timeUp: BOOL;
	fbresetTON: TON;
END_VAR
CASE state OF
1:
(*Receive information*)
	fbReceiveTON(  IN := FALSE, PT:=T#0s); (*Receive first request immediately*)
	fbReceiveTON(  IN := TRUE ); (*Start a timer to ensure complete transfer of information*)

		IF fbReceiveTON.Q THEN
			fbReceiveTON(  IN := FALSE);
			fb_receive(bExecute:=FALSE);  (*Generate a rising edge to start receiving data*)
			fb_receive
			(
				sSrvNetId:='',
				hSocket :=socketToUse,
				cbLen:=SIZEOF(receiveBuffer)-cbReceived,
				pDest:=ADR(receiveBuffer)+cbReceived,
				tTimeout:=T#5s,
				nRecBytes=>bytesReceived,
				nErrId=>receiveError,
				bExecute:=TRUE,
			);

	(*Move to the receive completion state*)
	state:=2;
	END_IF

2:
(*Continue receiving data*)
	fb_receive( bExecute := FALSE );
	IF NOT fb_receive.bBusy THEN
		IF NOT fb_receive.bError THEN (*If no error has occurred then start the actual receiving of data*)

			IF (fb_receive.nRecBytes>0) THEN (*Bytes have been received*)

				startPos:=cbReceived; (*index of first data byte*)
				endPos:=cbReceived+fb_receive.nRecBytes-1; (*index of last byte*)
				cbReceived:=cbReceived+fb_receive.nRecBytes; (*Calculating the number of received data bytes*)
				cbFrame:=0; (*Reset the frame length*)


				IF cbReceived<SIZEOF(sFromClient) THEN (*no overflow*)
					fbReceiveTON(IN:=FALSE, PT:=T#0S);

					(*Search for the string delimiter(separation character for different strings)*)
					FOR idx:=startPos TO endPos BY 1 DO
						IF receiveBuffer[idx]=0 THEN (*String delimiter found*)
							cbFrame:=idx+1;(*calculate length of received string*)
							MEMCPY(ADR(sFromClient), ADR(receiveBuffer),cbFrame); (*copy the received string to the output variable*)
							MEMMOVE(ADR(receiveBuffer), ADR(receiveBuffer[cbFrame]), cbReceived-cbFrame);(*move remaining data bytes*)
							dataReceived:=TRUE;  	(*Send an acknowledgement of data received*)
							state:=3; (*Move to the receive completion state*)
							endFound:=TRUE;
							EXIT;
						END_IF
					END_FOR
				ELSE(*no more free buffer space-overflow*)

					dataReceived:=FALSE; (*Go to error state*)
					overflow:=TRUE;
					state:=4;
				END_IF
			ELSE(*no data received*)
					fbReceiveTON(IN:=FALSE, PT:=T#0ms);
					state:=1;
			END_IF
		ELSE(*error receiving data, exit function*)
			state:=4;
			dataReceived:=FALSE;
		END_IF
	END_IF

3:
	(*State used to process data*)
	botton:=(STRING_TO_LREAL(MID(sFromClient, 4, 1)));  (*Extract the x distance*)
IF(botton = 48) THEN
	xAxis:=((STRING_TO_LREAL(MID(sFromClient, 5, 5))-32768)/80);
	yAxis:=((STRING_TO_LREAL(MID(sFromClient, 5,10))-32768)/-80);
	zAxis:=((STRING_TO_LREAL(MID(sFromClient, 5, 15))-32768)/-80);
END_IF
IF(botton = 32)THEN
	yAxis:=((STRING_TO_LREAL(MID(sFromClient, 5, 5)))*40);
	xAxis:=((STRING_TO_LREAL(MID(sFromClient, 5,10)))*40);
	zAxis:=((STRING_TO_LREAL(MID(sFromClient, 5, 15)))*40);
END_IF

	fb_receive(bExecute:=FALSE); (*Reset the receive function*)
	startPos:=0; (*reset buffer beginning pointer*)
	endPos:=0;  (*reset buffer end pointer*)
	cbReceived:=0; (*reset bytes received counter*)
	sFromClient:=''; (*reset transition variable*)


	state:=1;
	RETURN;

4: (*Unused except for as an error state*)
trigger1:=FALSE; trigger2:=TRUE;  timerOn:=TRUE;(* reset arduino*)
fbresetTON(IN:=timerOn, PT:=REAL_TO_TIME(100), Q=>timeUp, ET=>);

IF (timeUp=TRUE)  THEN
trigger2:=FALSE;
timerOn:=FALSE;
END_IF

	(*Clear buffer-PROBABLY UNNECESSARY*)

	receiveBuffer[0]:=0;
	receiveBuffer[1]:=0;
	receiveBuffer[2]:=0;
	receiveBuffer[3]:=0;
	receiveBuffer[4]:=0;
	receiveBuffer[5]:=0;
	receiveBuffer[6]:=0;
	receiveBuffer[7]:=0;
	receiveBuffer[8]:=0;
	receiveBuffer[9]:=0;
	receiveBuffer[10]:=0;
	receiveBuffer[11]:=0;
	receiveBuffer[12]:=0;
	receiveBuffer[13]:=0;
	receiveBuffer[14]:=0;
	receiveBuffer[15]:=0;
receiveBuffer[16]:=0;
receiveBuffer[17]:=0;
receiveBuffer[18]:=0;
receiveBuffer[19]:=0;


	state:=1;


END_CASE;
END_FUNCTION_BLOCK

(* POU MainFast, ST *)
PROGRAM MainFast
VAR
	fblocalization:  localization;
END_VAR
fblocalization();
END_PROGRAM

(* POU localization, ST *)
FUNCTION_BLOCK localization  (* to be call by fb movement only*)  (* calls  fb kalman filter*)
VAR
	w1: LREAL;
	w2: LREAL;
	w3: LREAL;
	w4: LREAL;
	sw1: LREAL;
	sw2: LREAL;
	sw3: LREAL;
	sw4: LREAL;
	encoder1: AXIS_REF;
	encoder2: AXIS_REF;
	encoder3: AXIS_REF;
	encoder4: AXIS_REF;
	globalePosX: LREAL;
	globalePosY: LREAL;
	heading_radians1: LREAL;
	globalePosX1: LREAL;
	globalePosY1: LREAL;
	sencoderX: ARRAY[1..5] OF		LREAL;
	sencoderY: ARRAY[1..5] OF		LREAL;
	sheading: ARRAY[1..5] OF		LREAL;
	fbkalmanFilter: ARRAY[1..3] OF 	kalmanFilter;
	fbekalmanFilter: ARRAY[1..3] OF 	extendedKalmanFilter;
	fbTON3: TON;
	startTimer3: BOOL;
	timer3On: BOOL;
	A: LREAL;
	q: INT;
	differentX: LREAL;
	differentY: LREAL;
	arduinoCalculate1: arduinoCalculation;
	xDistA: LREAL;
	yDistA: LREAL;
	combinedXOld: LREAL := 0;
	combinedYOld: LREAL := 0;
	combinedHOld: LREAL := 0;
	count: INT;
	velocityX: LREAL;
	velocityY: LREAL;
	velocityH: LREAL;
	heading_radians: LREAL;
	combinedXOld1: LREAL;
	combinedYOld1: LREAL;
	combinedHOld1: LREAL;
	velocityX1: LREAL;
	velocityY1: LREAL;
	velocityH1: LREAL;
	moveA: BOOL;
	v4: LREAL;
	v3: LREAL;
	v: LREAL;
	v1: LREAL;
	v2: LREAL;
	ow1: LREAL;
	ow2: LREAL;
	ow3: LREAL;
	ow4: BOOL;
	dx: LREAL;
	dy: LREAL;
	dh: LREAL;
	x: LREAL;
	h: LREAL;
	y: LREAL;
	ox: LREAL;
	oy: LREAL;
	oh: LREAL;
	hr: LREAL;
	vx: LREAL;
	vy: LREAL;
	vh: LREAL;
END_VAR
(* from wheel motor encoder*)
w1:=axis1.NcToPlc.ActPos;
w2:=-axis2.NcToPlc.ActPos;
w3:=axis3.NcToPlc.ActPos;
w4:=-axis4.NcToPlc.ActPos;
encoderY[3]:=0.025*((w1-sw1)+(w2-sw2)+(w3-sw3)+(w4-sw4))*1.634*1.006;
encoderX[3]:=-0.025*((w1-sw1)-(w2-sw2)-(w3-sw3)+(w4-sw4))*1.339*1.006;
heading[3]:=(-0.025*(-(w1-sw1)+(w2-sw2)-(w3-sw3)+(w4-sw4))*0.144);

(* set ALL to zero at start of motion*)
IF (home) THEN
sencoderX[5]:=0.0;
sencoderX[1]:=encoder1.NcToPlc.ActPos*COS(10/180*3.142)-encoder2.NcToPlc.ActPos*SIN(10/180*3.142);
sencoderX[2]:=encoder3.NcToPlc.ActPos*COS(10/180*3.142)-encoder4.NcToPlc.ActPos*SIN(10/180*3.142);
xDistA:=0;
yDistA:=0;
sencoderX[4]:=0;
sencoderY[4]:=0;
sencoderY[5]:=0.0;
sencoderY[1]:=encoder1.NcToPlc.ActPos*SIN(10/180*3.142)+encoder2.NcToPlc.ActPos*COS(10/180*3.142);
sencoderY[2]:=encoder3.NcToPlc.ActPos*SIN(10/180*3.142)+encoder4.NcToPlc.ActPos*COS(10/180*3.142);
heading[1]:=0.0;
sheading[4]:=headingA;
sw1:=axis1.NcToPlc.ActPos;
sw2:=-axis2.NcToPlc.ActPos;
sw3:=axis3.NcToPlc.ActPos;
sw4:=-axis4.NcToPlc.ActPos;
globalePosX:=0;
globalePosY:=0;
x:=0;
y:=0;
h:=0;
home:=FALSE;
END_IF

(* continue to read data*)
	encoderX[1]:=(encoder1.NcToPlc.ActPos*COS(10/180*3.142)-encoder2.NcToPlc.ActPos*SIN(10/180*3.142) - sencoderX[1]);
	encoderY[1]:=(encoder1.NcToPlc.ActPos*SIN(10/180*3.142)+encoder2.NcToPlc.ActPos*COS(10/180*3.142) - sencoderY[1]);

	encoderX[2]:=(encoder3.NcToPlc.ActPos*COS(10/180*3.142)-encoder4.NcToPlc.ActPos*SIN(10/180*3.142) - sencoderX[2]);
	encoderY[2]:=(encoder3.NcToPlc.ActPos*SIN(10/180*3.142)+encoder4.NcToPlc.ActPos*COS(10/180*3.142) - sencoderY[2]);


(*Heading1 calculation from encoder 2 and 3, assume encoder 2 at origin*)
	differentX:=encoderX[2]-encoderX[1]-0.1;
	differentY:=encoderY[2]-encoderY[1]+550;

	IF (differentX>=0 AND differentY>=0) THEN A:=ATAN(differentY/differentX)*180/3.142; heading[1]:=180-(A-(0.03)); Q:=1; 		(* 1st quad*)
	ELSIF (differentX<0 AND differentY>=0) THEN A:=ATAN(differentY/-differentX)*180/3.142;heading[1]:=180-(180-A-(0.03)); Q:=2;  (* 2nd quad*)
	ELSIF (differentX<0 AND differentY<0) THEN A:=ATAN(differentY/differentX)*180/3.142; heading[1]:=180-(180+A-(0.03));    Q:=3;	(* 3rd quad*)
	ELSIF (differentX>=0 AND differentY<0) THEN A:=ATAN(-differentY/differentX)*180/3.142; heading[1]:=180-(360-A-(0.03)); Q:=4;   	(* 4th quad*)
	END_IF
IF heading[1] < -180 THEN heading[1]:=heading[1]+360; END_IF
IF heading[1] > 180 THEN heading[1]:=heading[1]-360;   END_IF(* heading is always between +180 to -180*)

(* arduino*)
	arduinoCalculate1(xDistA=>xDistA, yDistA=>ydistA);
	encoderX[4]:=xDistA;
	encoderY[4]:=yDistA;
	heading[4]:=headingA-sheading[4]+90;
	IF (heading[4]>360) THEN heading[4]:=heading[4]-360; END_IF
	IF (heading[4]<-360) THEN heading[4]:=heading[4]+360; END_IF
IF (trigger1=TRUE AND moveA=FALSE) THEN moveA:= TRUE; END_IF
IF (trigger3=FALSE AND moveA=TRUE) THEN sencoderX[4]:=encoderX[4];sencoderY[4]:=encoderY[4];moveA:=FALSE; END_IF

(*kalman filter.   cycle time = 10 ms*)
(*IF (trigger3=TRUE AND timer3On=FALSE) THEN*)
fbTON3(IN:=startTimer3, PT:=LREAL_TO_TIME(50) , Q=>timer3On);
count:=count+1;
IF (count>0) THEN startTimer3:=TRUE; END_IF
	IF (timer3On=TRUE) THEN
	timer3On:=FALSE;
	startTimer3:=FALSE;
	count:=0;
(* weighted average to combine the spherical ball encoder [2] to the wheel position encoder[3] combined signal =[5]*)
	encoderX[5]:=0.4*encoderX[2]+0.6*encoderX[3];
	encoderY[5]:=encoderY[3];
	fbkalmanFilter[3](reading:=(heading[1]-heading[3]),target:=0,noiseVar:= 0.1);
	heading[5]:=fbkalmanFilter[3].out+heading[3];
(*convert to world before arduino*)
	heading_radians1 :=  heading[5]/180 * 3.1415963;
	globalePosX1 := globalePosX1 + SIN(heading_radians1) *( encoderX[5] -combinedXOld1) +  COS(heading_radians1) * (encoderY[5] - combinedYOld1);
	globalePosY1 := globalePosY1 + SIN(heading_radians1) * (encoderY[5] - combinedYOld1) - COS(heading_radians1) *( encoderX[5] -combinedXOld1);
	velocityX1:=(encoderX[5]-combinedXOld1)/0.05;
	velocityY1:=(encoderY[5]-combinedYOld1)/0.05;
	velocityH1:=(combinedH-combinedHOld1)/0.05;

	combinedXOld1:=encoderX[5];
	combinedYOld1:=encoderY[5];
	combinedHOld1:=heading[5];

(*arduino KF*)
	fbekalmanFilter[1](reading:=(encoderX[4]-encoderX[5]),target:=0,noiseVar:= 0.1);
	combinedX:=fbekalmanFilter[1].out+encoderX[5];
	fbekalmanFilter[2](reading:=(encoderY[4]-encoderY[5]),target:=0,noiseVar:= 0.1);
	combinedY:=fbekalmanFilter[2].out+encoderY[5];
	fbekalmanFilter[3](reading:=(heading[4]-heading[5]),target:=0,noiseVar:= 0.1);
	combinedH:=fbekalmanFilter[3].out+heading[5];

(*	velocityX:=(combinedX-combinedXOld)/0.05;
	velocityY:=(combinedY-combinedYOld)/0.05;
	velocityH:=(combinedH-combinedHOld)/0.05;*)

(*convert to world (after arduino) *)
	heading_radians :=  combinedH/180 * 3.1415963;
	globalePosX := globalePosX + SIN(heading_radians) *(combinedX - combinedXOld) +  COS(heading_radians) * (combinedY - combinedYOld);
	globalePosY := globalePosY + SIN(heading_radians) * (combinedY - combinedYOld) - COS(heading_radians) *( combinedX - combinedXOld);

	combinedXOld:=combinedX;
	combinedYOld:=combinedY;
	combinedHOld:=combinedH;

	END_IF

dx:=combinedX-ox;
dy:=combinedY-oy;
dh:=combinedH-oh;
hr := h/180 * 3.1415963;

x := x + dx*SIN(hr) + dy*COS(hr);
y := y + dx*COS(hr) - dy*SIN(hr);
h := h+dh;
IF (h > 360) THEN
	h := h - 360;
END_IF
IF (h < -360) THEN
	h := h + 360;
END_IF

ox:=combinedX;
oy:=combinedY;
oh:=combinedH;

v1:=axis1.NcToPlc.ActVelo;
v2:=-axis2.NcToPlc.ActVelo;
v3:=axis3.NcToPlc.ActVelo;
v4:=-axis4.NcToPlc.ActVelo;

velocityX:=0.025*((v1)+(v2)+(v3)+(v4))*1.634*1.006;
velocityY:=-0.025*((v1)-(v2)-(v3)+(v4))*1.339*1.006;
velocityH:=-0.025*(-(v1)+(v2)-(v3)+(v4))*0.144;

vx := velocityX*SIN(hr) + velocityY*COS(hr);
vy := velocityX*COS(hr) - velocityY*SIN(hr);
vh := velocityH;

(*output
robotPosTheta:=combinedH;
robotPosX:=globalePosX1;
robotPosY:=globalePosY1;
robotVelX:=velocityX1;
robotVelY:=velocityY1;
robotVelTheta:=velocityH;*)

LOCrobotPosX:=y;
LOCrobotPosY:=x;
LOCrobotPosTheta:=h;
LOCrobotVelX:=vx;
LOCrobotVelY:=vy;
LOCrobotVelTheta:=vh;
RETURN;
END_FUNCTION_BLOCK

(* POU kalmanFilter, ST *)
FUNCTION_BLOCK kalmanFilter
VAR_INPUT
	reading: LREAL;
	target: LREAL;
	noiseVar: LREAL;
END_VAR
VAR_OUTPUT
	out: LREAL;
END_VAR
VAR
	control: LREAL;
	oldP: LREAL;
	newP: LREAL := 1.0;
	oldX: LREAL;
	newX: LREAL:=0.0;
	K: LREAL;
	oldPredict: LREAL:=0.0;

END_VAR
control:=target-NewX;
(* timeupdate*)

oldP :=newP;
oldX:=newX+control;

(*measurement update*)

K:=oldP / (oldP+noiseVar);
NewX:=oldX+K*(reading-oldX);
newP:=(1-K)*oldP;
out:=NewX;

RETURN;
END_FUNCTION_BLOCK

(* POU extendedKalmanFilter, ST *)
FUNCTION_BLOCK extendedKalmanFilter
VAR_INPUT
	reading: LREAL;
	target: LREAL;
	noiseVar: LREAL;
END_VAR
VAR_OUTPUT
	out: LREAL;
END_VAR
VAR
	control: LREAL;
	estP: LREAL;
	newP: LREAL := 1.0;
	estX: LREAL;
	newX: LREAL:=0.0;
	newK: LREAL;
	oldPredict: LREAL:=0.0;
	count:INT;

(*extened KF*)
	F: LREAL:=1.0;
	H: LREAL:=1.0;
	oldfuncH: LREAL;
	funcH:LREAL;
	oldfuncF: LREAL;
	funcF: LREAL;
	oldX: LREAL;
	oldestX: LREAL;
END_VAR
(*kalman filter.   cycle time = 10 ms;   added f and h for extended KF assume B = 1*)
control:=target-NewX;
count:=count+1;

(* timeupdate*)
oldfuncF:=funcF;
funcF:=F*newX;
IF (newX-oldX<>0) THEN F:=(funcF-oldfuncF)/(newX-oldX); END_IF
estP :=F*newP*F;  (* assume Q =0 *)
oldestX:=estX;
estX:=funcF+control;

(*measurement update*)
newK:=H*estP / (H*estP*H+noiseVar);

oldfuncH:=funcH;
funcH:=H*estX;
IF (estX-oldestX<>0) THEN H:=(funcH-oldfuncH)/(estX-oldestX); END_IF
oldX:=newX;
newX:=estX+newK*(reading-funcH);
newP:=(1-newK*H)*estP;
out:=NewX;

RETURN;
END_FUNCTION_BLOCK

(* POU arduinoCalculation, ST *)
FUNCTION_BLOCK arduinoCalculation
VAR_INPUT

END_VAR
VAR_OUTPUT
	xDistA: LREAL;
	yDistA: LREAL;

END_VAR
VAR
	connectArduino1:				ArduinoConnect;
	disconnectArduino1:			ArduinoDisconnect;
	receiveData1:				ArduinoReceiveData;

	tcpSocket: T_HSOCKET;
	connectionOpen: BOOL:=FALSE;
	closeConnection: BOOL:=TRUE;
	dataReceived: BOOL;
	heading: LREAL;
	xAccA: ARRAY[1..10] OF LREAL;
	yAccA: ARRAY[1..10] OF LREAL;
	xVelA: ARRAY[1..3] OF LREAL;
	yVelA: ARRAY[1..3] OF LREAL;
	xVelB: ARRAY[1..3] OF LREAL;
	xBias: LREAL;
	yBias: LREAL;
	xAccel: LREAL;
	yAccel: LREAL;
	xVel:LREAL;
	yVel:LREAL;
	xPVel: LREAL:=0;
	yPVel:LREAL:=0;
	xPDist: LREAL;
	yPDist:LREAL;
	j: INT:=0;
	astart:BOOL;
	delayA: BOOL;
(*send to file*)
	n:INT:=0;
	fboutputToFile: outputToFile2;
	sent1: BOOL:=FALSE;
	delayB: BOOL;
	error: BOOL;
(*calculate velocity*)
	step:UINT:=0;
	i:UINT;
	calA:UINT:=55;
	calB:UINT:=30;
	sendAve: INT:=4;
	k: UINT:=0;
	velWheelX: LREAL;
	w1: LREAL;
	sw1: LREAL;
	w2: LREAL;
	sw2: LREAL;
	w3: LREAL;
	sw3: LREAL;
	w4: LREAL;
	sw4: LREAL;
	wheelVelY: LREAL;
	wheelVelX: LREAL;
	fbekalmanFilter:	ARRAY[1..2] OF 	extendedKalmanFilter;
	xVelk: LREAL;
	yVelK: LREAL;

	ybiasAcc: LREAL;
	xbiasAcc: LREAL;
	ybiasAccP: LREAL;
	xbiasAccP: LREAL;
	xDistAk: LREAL;
	yDistAk: LREAL;
	xPDistk: LREAL;
	yPDistk: LREAL;
END_VAR
(*Arduino*)
(*Close TCP port from last time-remove after DEBUG*)
IF closeConnection THEN
	disconnectArduino1(bCloseAll:=closeConnection);
	closeConnection:=FALSE;
END_IF

(*Open a connection*)
IF (connectionOpen=FALSE) THEN
	connectArduino1(arduinoConnected=>connectionOpen, socketToUse=>tcpSocket);
END_IF

IF (connectionOpen=TRUE) THEN
receiveData1(socketToUse:=tcpSocket,);
xAccel:=receiveData1.xAccel*calA;
yAccel:=receiveData1.yAccel*calB;
END_IF


(* Calculation*)
IF reset THEN
FOR i:=1 TO 10 BY 1 DO xAccA[1]:=0;	yAccA[i]:=0; END_FOR
		xBias:=0; 		yBias:=0;
		xAccel:=0; 		yAccel:=0;
		xVel:=0;  		yVel:=0;
		xPVel:=0; 		yPVel:=0;
		xPDist:=0; 		yPDist:=0;
		j:=0; k:=0;
		astart:=FALSE; 		delayA:=FALSE;
		sw1:=0;sw2:=0;sw3:=0;sw4:=0;
		step:=0;
END_IF
(* from wheel motor encoder*)
w1:=axis1.NcToPlc.ActVelo;
w2:=-axis2.NcToPlc.ActVelo;
w3:=axis3.NcToPlc.ActVelo;
w4:=-axis4.NcToPlc.ActVelo;
wheelVelY:=0.025*((w1-sw1)+(w2-sw2)+(w3-sw3)+(w4-sw4))*1.634*1.006/1000;
wheelVelX:=-0.025*((w1-sw1)-(w2-sw2)-(w3-sw3)+(w4-sw4))*1.339*1.006/1000;

(*from inertia sensor*)
IF (xAccel<>xAccA[1]) OR (yAccel<>yAccA[1])THEN
	dataReceived:=TRUE;
END_IF  (*use acceleration data to check the change in data as a new input*)

IF (trigger1=TRUE OR k>0 ) THEN trigger3:=TRUE; ELSE trigger3:=FALSE;  END_IF

IF dataReceived THEN
	dataReceived := FALSE;
	xAccA[1]:= xAccel; yAccA[1]:=yAccel;
	ybiasAcc:=(yAccel-yBias);
	xbiasAcc:=(xAccel-xBias);

CASE step OF
	0:	(* calculate the bias when not moving*)
		IF (trigger3=FALSE ) THEN
		xAccA[10]:= xAccA[9]; yAccA[10]:=yAccA[9];
		xAccA[9]:= xAccA[8]; yAccA[9]:=yAccA[8];
		xAccA[8]:= xAccA[7]; yAccA[8]:=yAccA[7];
		xAccA[7]:= xAccA[6]; yAccA[7]:=yAccA[6];
		xAccA[6]:= xAccA[5]; yAccA[6]:=yAccA[5];
		xAccA[5]:= xAccA[4]; yAccA[5]:=yAccA[4];
		xAccA[4]:= xAccA[3]; yAccA[4]:=yAccA[3];
		xAccA[3]:= xAccA[2]; yAccA[3]:=yAccA[2];
		xAccA[2]:= xAccA[1]; yAccA[2]:=yAccA[1];
		xBias:=(xAccA[1]+xAccA[2]+xAccA[3]+xAccA[4]+xAccA[5]+xAccA[6]+xAccA[7]+xAccA[8]+xAccA[9]+xAccA[10])/10;
		yBias:=(yAccA[1]+yAccA[2]+yAccA[3]+yAccA[4]+yAccA[5]+yAccA[6]+yAccA[7]+yAccA[8]+yAccA[9]+yAccA[10])/10;
		k:=0;
		ELSE (* acceleration starts*)
		astart:=TRUE;
		(*xVelA[1]:=xVelA[1]+(xbiasAcc+xbiasAccP)/2*0.01*sendAve; 		yVelA[1]:=yVelA[1]+(ybiasAcc+ybiasAccP)/2*0.01*sendAve;*)
		xVelA[1]:=xVelA[1]+COS(heading*3.142/180)*(xbiasAcc+xbiasAccP)/2*0.01*sendAve+SIN(heading*3.142/180)*(ybiasAcc+ybiasAccP)/2*0.01*sendAve;
		yVelA[1]:=yVelA[1]+SIN(heading*3.142/180)*(xbiasAcc+xbiasAccP)/2*0.01*sendAve+COS(heading*3.142/180)*(ybiasAcc+ybiasAccP)/2*0.01*sendAve;
		K:=K+1;
		step := 1;
		END_IF
	1:(* Acceleration *)
		IF (xbiasAcc<0.1 AND xbiasAcc>-0.1) THEN xbiasAcc:=0; END_IF
		IF (ybiasAcc<0.1 AND ybiasAcc>-0.1) THEN xbiasAcc:=0; END_IF
		IF(trigger2=FALSE ) THEN
(*		xVelA[1]:=xVelA[1]+(xbiasAcc+xbiasAccP)/2*0.01*sendAve; 		yVelA[1]:=yVelA[1]+(ybiasAcc+ybiasAccP)/2*0.01*sendAve;*)
		xVelA[1]:=xVelA[1]+COS(heading*3.142/180)*(xbiasAcc+xbiasAccP)/2*0.01*sendAve+SIN(heading*3.142/180)*(ybiasAcc+ybiasAccP)/2*0.01*sendAve;
		yVelA[1]:=yVelA[1]+SIN(heading*3.142/180)*(xbiasAcc+xbiasAccP)/2*0.01*sendAve+COS(heading*3.142/180)*(ybiasAcc+ybiasAccP)/2*0.01*sendAve;
		K:=K+1;
		ELSE(* add one more point *)
(*		xVelA[1]:=xVelA[1]+(xbiasAcc+xbiasAccP)/2*0.01*sendAve; 		yVelA[1]:=yVelA[1]+(ybiasAcc+ybiasAccP)/2*0.01*sendAve;*)
		xVelA[1]:=xVelA[1]+COS(heading*3.142/180)*(xbiasAcc+xbiasAccP)/2*0.01*sendAve+SIN(heading*3.142/180)*(ybiasAcc+ybiasAccP)/2*0.01*sendAve;
		yVelA[1]:=yVelA[1]+SIN(heading*3.142/180)*(xbiasAcc+xbiasAccP)/2*0.01*sendAve+COS(heading*3.142/180)*(ybiasAcc+ybiasAccP)/2*0.01*sendAve;
		K:=K+1;
		step:=2;
		END_IF
	2:	(*add one more acc because of the time delay due to mov ave*)
		IF (xbiasAcc<0.1 AND xbiasAcc>-0.1) THEN xbiasAcc:=0; END_IF
		IF (ybiasAcc<0.1 AND ybiasAcc>-0.1) THEN xbiasAcc:=0; END_IF
		(*xVelA[1]:=xVelA[1]+(xbiasAcc+xbiasAccP)/2*0.01*sendAve; 		yVelA[1]:=yVelA[1]+(ybiasAcc+ybiasAccP)/2*0.01*sendAve;*)
		xVelA[1]:=xVelA[1]+COS(heading*3.142/180)*(xbiasAcc+xbiasAccP)/2*0.01*sendAve+SIN(heading*3.142/180)*(ybiasAcc+ybiasAccP)/2*0.01*sendAve;
		yVelA[1]:=yVelA[1]+SIN(heading*3.142/180)*(xbiasAcc+xbiasAccP)/2*0.01*sendAve+COS(heading*3.142/180)*(ybiasAcc+ybiasAccP)/2*0.01*sendAve;
		IF (trigger2=FALSE AND trigger1=TRUE) THEN step:= 1; ELSE step:=3; END_IF
		IF (trigger1= FALSE) THEN step:=4; END_IF

	3:	(* constant velocity *)
		IF (trigger2=TRUE AND trigger1=TRUE) THEN step:= 3; ELSE
			IF (trigger1= FALSE) THEN step:=4; ELSE step:=1; END_IF
		END_IF
		xVelA[1]:=xPVel; 				yVelA[1]:=yPVel;
	4:(* Deceleration add one more data*)
		IF (xbiasAcc<0.1 AND xbiasAcc>-0.1) THEN xbiasAcc:=0; END_IF
		IF (ybiasAcc<0.1 AND ybiasAcc>-0.1) THEN xbiasAcc:=0; END_IF
		(*xVelA[1]:=xVelA[1]+(xbiasAcc+xbiasAccP)/2*0.01*sendAve; 		yVelA[1]:=yVelA[1]+(ybiasAcc+ybiasAccP)/2*0.01*sendAve;*)
		xVelA[1]:=xVelA[1]+COS(heading*3.142/180)*(xbiasAcc+xbiasAccP)/2*0.01*sendAve+SIN(heading*3.142/180)*(ybiasAcc+ybiasAccP)/2*0.01*sendAve;
		yVelA[1]:=yVelA[1]+SIN(heading*3.142/180)*(xbiasAcc+xbiasAccP)/2*0.01*sendAve+COS(heading*3.142/180)*(ybiasAcc+ybiasAccP)/2*0.01*sendAve;
		K:=K-1;
		step:=5;
	5:(* Deceleration*)
		IF (trigger1= FALSE) THEN step:=5;ELSE k:=0; step:=1; END_IF
		IF (k>0) THEN
			IF (k>10) THEN k:=10; END_IF
			IF (xbiasAcc<0.1 AND xbiasAcc>-0.1) THEN xbiasAcc:=0; END_IF
			IF (ybiasAcc<0.1 AND ybiasAcc>-0.1) THEN xbiasAcc:=0; END_IF
		(*xVelA[1]:=xVelA[1]+(xbiasAcc+xbiasAccP)/2*0.01*sendAve; 		yVelA[1]:=yVelA[1]+(ybiasAcc+ybiasAccP)/2*0.01*sendAve;*)
		xVelA[1]:=xVelA[1]+COS(heading*3.142/180)*(xbiasAcc+xbiasAccP)/2*0.01*sendAve+SIN(heading*3.142/180)*(ybiasAcc+ybiasAccP)/2*0.01*sendAve;
		yVelA[1]:=yVelA[1]+SIN(heading*3.142/180)*(xbiasAcc+xbiasAccP)/2*0.01*sendAve+COS(heading*3.142/180)*(ybiasAcc+ybiasAccP)/2*0.01*sendAve;
		k:=K-1;
		ELSE
		step:= 0;
		xbiasAcc:=0; 		ybiasAcc:=0;
		xbiasAccP:=0; 	ybiasAccP:=0;
		xAccel:=0; 		yAccel:=0;
		xVelA[1]:=0;  		yVelA[1]:=0;
		xPVel:=0; 		yPVel:=0;
		END_IF
	END_CASE
ybiasAccP:=ybiasAcc;  xbiasAccP:=xBiasAcc;
(*alt method using if*)(*
	IF (trigger3=FALSE) THEN  (* calculate the bias*)
	step:= 0;
	xVelA[1]:=0;  		yVelA[1]:=0;
	xPVel:=0; 		yPVel:=0;
	xAccA[10]:= xAccA[9]; yAccA[10]:=yAccA[9];
	xAccA[9]:= xAccA[8]; yAccA[9]:=yAccA[8];
	xAccA[8]:= xAccA[7]; yAccA[8]:=yAccA[7];
	xAccA[7]:= xAccA[6]; yAccA[7]:=yAccA[6];
	xAccA[6]:= xAccA[5]; yAccA[6]:=yAccA[5];
	xAccA[5]:= xAccA[4]; yAccA[5]:=yAccA[4];
	xAccA[4]:= xAccA[3]; yAccA[4]:=yAccA[3];
	xAccA[3]:= xAccA[2]; yAccA[3]:=yAccA[2];
	xAccA[2]:= xAccA[1]; yAccA[2]:=yAccA[1];
	xBias:=(xAccA[1]+xAccA[2]+xAccA[3]+xAccA[4]+xAccA[5]+xAccA[6]+xAccA[7]+xAccA[8]+xAccA[9]+xAccA[10])/10;
	yBias:=(yAccA[1]+yAccA[2]+yAccA[3]+yAccA[4]+yAccA[5]+yAccA[6]+yAccA[7]+yAccA[8]+yAccA[9]+yAccA[10])/10;
	xVel:=0; yVel:=0;	xDistA:=0; yDistA:=0;
	ELSE
	xVelA[1]:=xVelA[1]+(xbiasAcc+xbiasAccP)/2*0.01*sendAve; 		yVelA[1]:=yVelA[1]+(ybiasAcc+ybiasAccP)/2*0.01*sendAve;
	k:=k+1;
	END_IF

	IF (trigger1 =TRUE AND astart =FALSE) THEN astart:=TRUE;END_IF (*start*)

  	IF(trigger1 =TRUE AND trigger2=FALSE ) THEN  (*acceleration*)step:=1;
			IF (xbiasAcc<0.01 AND xbiasAcc>-0.01) THEN xbiasAcc:=0; END_IF
			IF (ybiasAcc<0.01 AND ybiasAcc>-0.01) THEN xbiasAcc:=0; END_IF
		IF(trigger2=FALSE ) THEN
		xVelA[1]:=xVelA[1]+(xbiasAcc+xbiasAccP)/2*0.01*sendAve; 		yVelA[1]:=yVelA[1]+(ybiasAcc+ybiasAccP)/2*0.01*sendAve;
		(*xDistA:=(xVel)*40+xDistA;  yDistA:=(yVel)*40+yDistA;*)
		k:=k+1;
		END_IF
	END_IF

	IF(trigger1 =TRUE AND trigger2=TRUE ) THEN (*constant velocity*)step:=2;
		IF (delayA=FALSE) THEN
		xVelA[1]:=xVelA[1]+(xbiasAcc+xbiasAccP)/2*0.01*sendAve; 		yVelA[1]:=yVelA[1]+(ybiasAcc+ybiasAccP)/2*0.01*sendAve;
		(*xDistA:=(xVel)*40+xDistA;  yDistA:=(yVel)*40+yDistA;*)
		k:=k+1;
		delayA:=TRUE;
			IF astart=TRUE THEN xPVel := xVel; yPVel:=yVel;END_IF  (*acceleration stage when astart is true*)
		ELSE
			xVelA[1]:=xPVel;yVelA[1]:=yPVel;
			xDistA:=(xVel)*40+xDistA;  yDistA:=(yVel)*40+yDistA;
		END_IF
	END_IF

	IF(trigger1 =FALSE AND trigger3=TRUE AND astart=TRUE) THEN  (*deceleration*)step:=3;
			IF (k>15) THEN k:=15; END_IF
		IF (k>0) THEN
			IF (xbiasAcc<0.01 AND xbiasAcc>-0.01) THEN xbiasAcc:=0; END_IF
			IF (ybiasAcc<0.01 AND ybiasAcc>-0.01) THEN xbiasAcc:=0; END_IF
		xVelA[1]:=xVelA[1]+(xbiasAcc+xbiasAccP)/2*0.01*sendAve; 		yVelA[1]:=yVelA[1]+(ybiasAcc+ybiasAccP)/2*0.01*sendAve;
		k:=K-1;
		END_IF
	END_IF

*)
	(* end of alt method*)
(* dist cal*)
	IF (xVelA[1]<0.001 AND xVelA[1]>-0.001) THEN xVelA[1]:=0; END_IF
	IF (yVelA[1]<0.002 AND yVelA[1]>-0.002) THEN yVelA[1]:=0; END_IF
	xPVel := xVelA[1]; 		yPVel:=yVelA[1];
	IF (trigger3) THEN
		xVel:=xVelA[1];
		yVel:=yVelA[1];
	ELSE
	xVel:=0;
	yVel:=0;
	END_IF

	(*fbekalmanFilter[1](reading:=(xVel-wheelVelX),target:=0,noiseVar:= 0.0035);    (* use wheel speed to KF with inertia sensor speed noise var need to vadify*)
	xVelk:=fbekalmanFilter[1].out+wheelVelX;
	fbekalmanFilter[2](reading:=(yVel-wheelVelY),target:=0,noiseVar:= 0.0035);
	yVelK:=fbekalmanFilter[2].out+wheelVelY;
	xDistAk:=(xVelk)*10*sendAve+xDistA;  					yDistAk:=(yVelk)*10*sendAve+yDistA;
	xPDistk:=xDistAk; 										yPDistk:=yDistAk;*)
	xDistA:=(xVel+xPVel)/2*10*sendAve+xDistA; 				yDistA:=(yVel+yPVel)/2*10*sendAve+yDistA;
	xPDist:=xDistA; 										yPDist:=yDistA;
(*for print to filedata*)
	IF(trigger3=TRUE AND n<=MAX_CSV_ROWS) THEN
	FILEDATA1[n,0]:=LREAL_TO_STRING(encoderX[2]);
	FILEDATA1[n,1]:=LREAL_TO_STRING(encoderY[2]);
	FILEDATA1[n,2]:=LREAL_TO_STRING(encoderX[3]);
	FILEDATA1[n,3]:=LREAL_TO_STRING(encoderY[3]);
	FILEDATA1[n,4]:=LREAL_TO_STRING(xDistA);
	FILEDATA1[n,5]:=LREAL_TO_STRING(yDistA);
	FILEDATA1[n,6]:=LREAL_TO_STRING(combinedX);
	FILEDATA1[n,7]:=LREAL_TO_STRING(combinedY);
	FILEDATA1[n,8]:=LREAL_TO_STRING(step);
	n:=n+1;(* end of print to filedata*)
	END_IF

END_IF (* end of data received*)
IF (trigger3=FALSE) THEN xDistA:=encoderX[3];yDistA:=encoderY[3];  END_IF

(* send data to file*)
IF ((astart=TRUE) AND (trigger3 = FALSE)) THEN sent1:=TRUE; astart:=FALSE;END_IF
fboutputToFile(database:=FILEDATA1,bWrite:=sent1,sFileName:= '\Hard Disk2\Temp\Acc7nov.csv');
sent1:=FALSE;

RETURN;
END_FUNCTION_BLOCK

(* POU ArduinoConnect, ST *)
FUNCTION_BLOCK ArduinoConnect
VAR


	(*Functions*)
	openSocket: BOOL:=FALSE;
	fb_listen: FB_SocketListen;
	fb_accept: FB_SocketAccept;
	(*Timers*)
	fbAcceptTON: TON;

	(*TCP socket variables*)
	activeSocketHandle: T_HSOCKET;
	socketHandle: T_HSOCKET;



	(*Error variables*)
	listenError: UDINT:=0;
	acceptError: UDINT;
	listenErrSet: BOOL;
	closeError: UDINT;
	sendError: UDINT;
	receiveError: UDINT;
	bSendError: BOOL;


	(*Trigger Variables*)
	bCloseAll: BOOL := TRUE;

	(*Connection information*)
	portNumber: INT:=8888;
	bAccepted: BOOL;

	(*Constants*)
	PLCPRJ_ACCEPT_POLLING_TIME: TIME:=T#1s;

	display: LREAL;
	heading: LREAL;

	state: INT:=0;

	xDist: LREAL;
	yDist: LREAL;
	zDist: LREAL;


	listening: BOOL;
	count: INT;
	fbresetTON: TON;
	timerOn: BOOL;
	timeUp: BOOL;
END_VAR
VAR_OUTPUT
	arduinoConnected: BOOL;
	socketToUse: T_HSOCKET;
END_VAR
CASE state OF
0:

IF(fb_Listen.hListener.localAddr.nPort=portNumber) THEN
RETURN;

ELSE
state:=1;
END_IF

1:
(*This code was built by Chris Jarrett, Auckland University, 2014. It is derived in part from the TCP/IP server example on www.beckhoff.com*)
(*Listening State*)
(*Open a connection*)
(*Create socket and check for errors*)

fb_listen
(
	sSrvNetId:='' ,
	sLocalHost:='',
	nLocalPort:=portNumber,
	bExecute:=TRUE,
	tTimeout:=T#5s,
	hListener=>socketHandle,
	nErrId=>listenError,
	bError=>listenErrSet,

);

	IF(fb_Listen.hListener.localAddr.nPort=portNumber) THEN
		fb_listen(bExecute:=FALSE); 		(*Start listening and move to the accept state*)

		state:=2;
	ELSE
		(*Return to the listening state*)
		state:=1;
	END_IF



2:

(*Start accepting a client connection*)
fbAcceptTON( IN := TRUE, PT := T#2s);  (*Start a timer to poll for the accepted connection*)
		IF fbAcceptTON.Q THEN
			fbAcceptTON( IN := FALSE );	(*Reset timer*)
			fb_accept(  bExecute := FALSE  ); (*Generate a rising edge to activate the accept function*)
			fb_accept(hListener := socketHandle, bExecute:= TRUE, hSocket=>activeSocketHandle );
			state:=3; (*Move to the state where the client is accepted*)

			fbAcceptTON( IN := FALSE);

		END_IF
3:
(*Complete accpeting the client connection*)
	fb_accept( bExecute := FALSE ); (*Reset the accept function to try connection again if necessary*)
	IF NOT fb_accept.bBusy THEN
		IF NOT fb_accept.bError THEN
			IF fb_accept.bAccepted THEN
				bAccepted := TRUE; (*If the client connection is accepted without error then move to the send state*)
				fb_accept(bExecute:=FALSE);
				socketToUse:=fb_accept.hSocket;

				state:=4;
			ELSE
				fb_listen(bExecute:=FALSE);
				fb_accept(bExecute:=FALSE);
				arduinoConnected:=FALSE; (*If the connection attempt was not successful, return the boolean as false*)
				fbAcceptTON( IN := FALSE);
				state:=2;

				END_IF
		END_IF
	END_IF
4:
arduinoConnected:=TRUE;
RETURN;

END_CASE;
END_FUNCTION_BLOCK

(* POU ArduinoDisconnect, ST *)
FUNCTION_BLOCK ArduinoDisconnect
VAR_INPUT
	bCloseAll: BOOL;
END_VAR
VAR_OUTPUT
	connectionClosed: BOOL;
END_VAR
VAR
	fb_closeAll: FB_SocketCloseAll;
END_VAR
(*This function closes the TCP/IP port being used the Arduino connection*)

IF bCloseAll THEN
	bCloseAll:=FALSE;
	(*Close all open ports*)
	fb_closeAll(sSrvNetId:='', bExecute:=TRUE, tTimeOut:=T#5s );
ELSE
	fb_closeAll(bExecute:=FALSE);
END_IF


(*Move to the listening state*)
IF NOT fb_closeAll.bError THEN
	connectionClosed:=TRUE;


ELSE
connectionClosed:=FALSE;
END_IF
RETURN;
END_FUNCTION_BLOCK

(* POU ArduinoReceiveData, ST *)
FUNCTION_BLOCK ArduinoReceiveData
VAR_INPUT
	socketToUse: T_HSOCKET;
END_VAR
VAR_OUTPUT
	dataReceived: BOOL;
	xAccel: LREAL;
	yAccel: LREAL;
END_VAR
VAR
	(*Connection timers*)
	fbReceiveTON: TON;

 	(*Functions*)
	fb_receive: FB_SocketReceive;

	(*Send and receive data and variables*)
	receiveBuffer: ARRAY[0..17] OF BYTE;
	bytesReceived: UDINT;
	sendBuffer: STRING;
	sendBufferAddress: DWORD;
	cbReceived, startPos, endPos, idx : UDINT;
	cbFrame: UDINT;
	sFromClient: T_MaxString;
	overflow: BOOL;
	endFound: BOOL;

	(*Error variables*)
	acceptError: UDINT;
	receiveError: UDINT;

	state: INT:=1;
	yDistString: STRING;
	xDistString: STRING;
	zDistString: STRING;
	headingString: STRING;
	timerOn: BOOL;
	timeUp: BOOL;
	fbresetTON: TON;
END_VAR
CASE state OF
1:
(*Receive information*)
	fbReceiveTON(  IN := FALSE, PT:=T#0s); (*Receive first request immediately*)
	fbReceiveTON(  IN := TRUE ); (*Start a timer to ensure complete transfer of information*)

		IF fbReceiveTON.Q THEN
			fbReceiveTON(  IN := FALSE);
			fb_receive(bExecute:=FALSE);  (*Generate a rising edge to start receiving data*)
			fb_receive
			(
				sSrvNetId:='',
				hSocket :=socketToUse,
				cbLen:=SIZEOF(receiveBuffer)-cbReceived,
				pDest:=ADR(receiveBuffer)+cbReceived,
				tTimeout:=T#5s,
				nRecBytes=>bytesReceived,
				nErrId=>receiveError,
				bExecute:=TRUE,
			);

	(*Move to the receive completion state*)
	state:=2;
	END_IF

2:
(*Continue receiving data*)
	fb_receive( bExecute := FALSE );
	IF NOT fb_receive.bBusy THEN
		IF NOT fb_receive.bError THEN (*If no error has occurred then start the actual receiving of data*)

			IF (fb_receive.nRecBytes>0) THEN (*Bytes have been received*)

				startPos:=cbReceived; (*index of first data byte*)
				endPos:=cbReceived+fb_receive.nRecBytes-1; (*index of last byte*)
				cbReceived:=cbReceived+fb_receive.nRecBytes; (*Calculating the number of received data bytes*)
				cbFrame:=0; (*Reset the frame length*)


				IF cbReceived<SIZEOF(sFromClient) THEN (*no overflow*)
					fbReceiveTON(IN:=FALSE, PT:=T#0S);

					(*Search for the string delimiter(separation character for different strings)*)
					FOR idx:=startPos TO endPos BY 1 DO
						IF receiveBuffer[idx]=0 THEN (*String delimiter found*)
							cbFrame:=idx+1;(*calculate length of received string*)
							MEMCPY(ADR(sFromClient), ADR(receiveBuffer),cbFrame); (*copy the received string to the output variable*)
							MEMMOVE(ADR(receiveBuffer), ADR(receiveBuffer[cbFrame]), cbReceived-cbFrame);(*move remaining data bytes*)
							dataReceived:=TRUE;  	(*Send an acknowledgement of data received*)
							state:=3; (*Move to the receive completion state*)
							endFound:=TRUE;
							EXIT;
						END_IF
					END_FOR
				ELSE(*no more free buffer space-overflow*)

					dataReceived:=FALSE; (*Go to error state*)
					overflow:=TRUE;
					state:=4;
				END_IF
			ELSE(*no data received*)
					fbReceiveTON(IN:=FALSE, PT:=T#1ms);
					state:=1;
			END_IF
		ELSE(*error receiving data, exit function*)
			state:=4;
			dataReceived:=FALSE;
		END_IF
	END_IF

3:
	(*State used to process data*)
	xAccel:=(STRING_TO_LREAL(MID(sFromClient, 6, 1)))/1000/16384*-9.8;  (*Extract the acceration*)
	yAccel:=(STRING_TO_LREAL(MID(sFromClient, 6, 7)))/1000/16384*9.8;
	headingA:=(STRING_TO_LREAL(MID(sFromClient, 4, 13)))/10;

	fb_receive(bExecute:=FALSE); (*Reset the receive function*)
	startPos:=0; (*reset buffer beginning pointer*)
	endPos:=0;  (*reset buffer end pointer*)
	cbReceived:=0; (*reset bytes received counter*)
	sFromClient:=''; (*reset transition variable*)

	state:=1;
	RETURN;

4: (*Unused except for as an error state*)
reset:=TRUE;

	(*Clear buffer-PROBABLY UNNECESSARY*)
	receiveBuffer[0]:=0;
	receiveBuffer[1]:=0;
	receiveBuffer[2]:=0;
	receiveBuffer[3]:=0;
	receiveBuffer[4]:=0;
	receiveBuffer[5]:=0;
	receiveBuffer[6]:=0;
	receiveBuffer[7]:=0;
	receiveBuffer[8]:=0;
	receiveBuffer[9]:=0;
	receiveBuffer[10]:=0;
	receiveBuffer[11]:=0;
	receiveBuffer[12]:=0;
	receiveBuffer[13]:=0;
	receiveBuffer[14]:=0;
	receiveBuffer[15]:=0;
receiveBuffer[16]:=0;
receiveBuffer[17]:=0;

	state:=1;


END_CASE;
END_FUNCTION_BLOCK

(* POU outputToFile2, ST *)
FUNCTION_BLOCK outputToFile2
VAR_INPUT
	database : ARRAY[0..MAX_CSV_ROWS, 0..MAX_CSV_COLUMNS ] OF STRING;
	bWrite			: BOOL := FALSE;(* Rising edge starts program execution *)
	sFileName	: T_MaxString;(* CSV destination file path and name *)
END_VAR
VAR_OUTPUT
END_VAR
(* Writing of CSV file in text mode. None of the field value is containing any non-printing control characters like line feed, carriage return, quotation marks, semicolon... *)
VAR
	sNetId			: T_AmsNetId := '';	(* TwinCAT system network address *)
	sCSVLine		: T_MaxString := '';(* Single CSV text line (row, record), we are using string as record buffer (your are able to see created fields) *)
	sCSVField		: T_MaxString := '';(* Single CSV field value (column, record field) *)
	bBusy			: BOOL;
	bError			: BOOL;
	nErrId			: UDINT;
	nRow	 		: UDINT 	:= 0;(* Row number (record) *)
	nColumn		: UDINT 	:= 0;(* Column number (record field) *)
	hFile			: UINT		:= 0;(* File handle of the source file *)
	step			: DWORD 	:= 0;
	fbFileOpen	: FB_FileOpen;(* Opens file *)
	fbFileClose	: FB_FileClose;(* Closes file *)
	fbFilePuts		: FB_FilePuts;(* Writes one record (line) *)
	fbWriter		: FB_CSVMemBufferWriter;(* Helper function block used to create CSV data bytes (single record line) *)

	(*database		: ARRAY[0..MAX_CSV_ROWS, 0..MAX_CSV_COLUMNS ] OF STRING(MAX_CSV_FIELD_LENGTH) := (* Source PLC database *)
	'0_0', '0_1', '0_2', '0_3', '0_4', '0_5',
	'1_0', '1_1', '1_2', '1_3', '1_4', '1_5',
	'2_0', '2_1', '2_2', '2_3', '2_4', '2_5',
	'3_0', '3_1', '3_2', '3_3', '3_4', '3_5',
	'4_0', '4_1', '4_2', '4_3', '4_4', '4_5',
	'5_0', '5_1', '5_2', '5_3', '5_4', '5_5';*)

END_VAR
CASE step OF
	0:	(* Wait for rising edge at bWrite variable *)
		IF bWrite THEN
			bWrite 		:= FALSE;
			bBusy 		:= TRUE;
			bError		:= FALSE;
			nErrId		:= 0;
			hFile		:= 0;
			nRow	 	:= 0;
			nColumn	:= 0;
			step 		:= 1;
		END_IF

	1:	(* Open source file *)
		fbFileOpen(  bExecute := FALSE  );
		fbFileOpen( 	sNetId := sNetId, sPathName := sFileName, nMode := FOPEN_MODEWRITE OR FOPEN_MODETEXT,(* Open file in TEXT mode! *)
						ePath := PATH_GENERIC, bExecute := TRUE );
		step := 2;

	2:(* Wait until open not busy *)
		fbFileOpen( bExecute := FALSE, bError => bError, nErrID => nErrID, hFile => hFile );
		IF NOT fbFileOpen.bBusy THEN
			IF NOT fbFileOpen.bError THEN
				step := 3;
			ELSE(* Error: file not found? *)
				step := 100;
			END_IF
		END_IF

	3:(* Convert one PLC record to CSV format *)
		sCSVLine := '';
		fbWriter.eCmd := eEnumCmd_First;(* Write first field value *)
		IF nRow <= MAX_CSV_ROWS THEN

			FOR nColumn := 0 TO MAX_CSV_COLUMNS BY 1 DO

				sCSVField := STRING_TO_CSVFIELD( database[ nRow, nColumn ], FALSE );(* TODO: Get field value from your application *)

				(* Add new field to the record buffer *)
				fbWriter( 	pBuffer := ADR( sCSVLine ), cbBuffer := SIZEOF( sCSVLine ) - 1, putValue := sCSVField, pValue := 0, cbValue := 0,
							bCRLF := ( nColumn = MAX_CSV_COLUMNS ) );(* bCRLF == TRUE => Write CRLF after the last field value *)
				IF fbWriter.bOk THEN
					fbWriter.eCmd := eEnumCmd_Next;(* Write next field value *)
				ELSE(* Error *)
					step := 100;
					RETURN;
				END_IF

			END_FOR(* FOR nColumn := 0... *)

			(* FB_FilePuts adds allready CR (carriage return) to the written line.
			We have to replace the $R$L characters with $L character to avoid double CR. *)
			IF RIGHT( sCSVLine, 2 ) = '$R$L' THEN
				sCSVLine := REPLACE( sCSVLine, '$L', 2, LEN( sCSVLine ) - 1 );
			END_IF

			nRow := nRow + 1;(* Increment number of created records (rows) *)
			step := 4;(* Write record to the file *)

		ELSE(* All rows written => Close file *)
			step := 10;
		END_IF

	4:	(* Write single text line *)
		fbFilePuts( bExecute := FALSE );
		fbFilePuts( sNetId := sNetId, hFile := hFile, sLine := sCSVLine, bExecute := TRUE );
		step := 5;

	5:(* Wait until write not busy *)
		fbFilePuts( bExecute := FALSE, bError => bError, nErrID => nErrID );
		IF NOT fbFilePuts.bBusy THEN
			IF NOT fbFilePuts.bError THEN
				step := 3;(* Write next record *)
			ELSE(* Error *)
				step := 100;
			END_IF
		END_IF

	10:	(* Close source file *)
		fbFileClose( bExecute := FALSE );
		fbFileClose( sNetId := sNetId, hFile := hFile, bExecute := TRUE );
		step := 11;

	11:(* Wait until close not busy *)
		fbFileClose( bExecute := FALSE, bError => bError, nErrID => nErrID );
		IF ( NOT fbFileClose.bBusy ) THEN
			hFile := 0;
			step := 100;
		END_IF

	100: (* Error or ready step => cleanup *)
		IF ( hFile <> 0 ) THEN
			step := 10; (* Close the source file *)
		ELSE
			bBusy := FALSE;
			step := 0;	(* Ready *)
		END_IF

END_CASE
END_FUNCTION_BLOCK

(* Visualisation MAINGUI
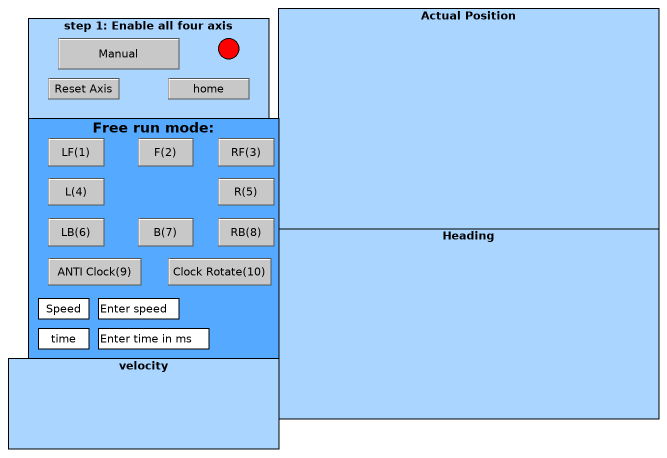
rectangle at (260,230)-(641,421): text "Heading"
rectangle at (10,20)-(251,121): text "step 1: Enable all four axis"
button at (40,40)-(161,71): text "Manual"; toggles MAIN.Manual
ellipse at (200,40)-(221,61): alarm colour if .trigger2
button at (30,80)-(101,101): text "Reset Axis"; taps reset
rectangle at (260,10)-(641,231): text "Actual Position"
rectangle at (10,120)-(261,451): text "Free run mode:"
button at (30,140)-(86,168): text "LF(1)"; taps MAIN.bMoveCombination[1]
button at (30,180)-(86,207): text "L(4)"; taps MAIN.bMoveCombination[4]
button at (30,220)-(86,248): text "LB(6)"; taps MAIN.bMoveCombination[6]
button at (120,140)-(175,168): text "F(2)"; taps MAIN.bMoveCombination[2]
button at (120,220)-(175,248): text "B(7)"; taps MAIN.bMoveCombination[7]
button at (200,140)-(256,168): text "RF(3)"; taps MAIN.bMoveCombination[3]
button at (200,180)-(256,207): text "R(5)"; taps MAIN.bMoveCombination[5]
button at (200,220)-(256,248): text "RB(8)"; taps MAIN.bMoveCombination[8]
button at (30,260)-(123,287): text "ANTI Clock(9)"; taps MAIN.bMoveCombination[9]
button at (150,260)-(253,287): text "Clock Rotate(10)"; taps MAIN.bMoveCombination[10]
rectangle at (80,330)-(191,351): text "Enter time in ms"; shows MAIN.timeToMoveReal; editable 0..20000
rectangle at (-10,360)-(261,451): text "velocity"
rectangle at (80,300)-(161,321): text "Enter speed"; shows MAIN.speedToMove; editable 0..2000
rectangle at (20,330)-(71,351): text "time"
rectangle at (20,300)-(71,321): text "Speed"
button at (150,80)-(231,101): text "home"; taps home
21 elements of other kinds (tables, trends, ...) not read
*)
